LIN {X 0,Y 560.526,Z 804.621,A -85,B 0,C 180,E1 21133.416,E2 21133.416} C_VEL
LIN {X 0,Y 560.837,Z 791.782,A -85,B 0,C 180,E1 21131.497,E2 21131.497} C_VEL
LIN {X 0,Y 561.234,Z 777.649,A -85,B 0,C 180,E1 21129.671,E2 21129.671} C_VEL
LIN {X 0,Y 561.729,Z 761.82,A -85,B 0,C 180,E1 21127.907,E2 21127.907} C_VEL
LIN {X 0,Y 562.275,Z 745.057,A -85,B 0,C 180,E1 21126.303,E2 21126.303} C_VEL
LIN {X 0,Y 562.895,Z 726.381,A -85,B 0,C 180,E1 21124.766,E2 21124.766} C_VEL
LIN {X 0,Y 563.513,Z 707.517,A -85,B 0,C 180,E1 21123.439,E2 21123.439} C_VEL
LIN {X 0,Y 564.133,Z 687.731,A -85,B 0,C 180,E1 21122.273,E2 21122.273} C_VEL
LIN {X 0,Y 564.708,Z 667.025,A -85,B 0,C 180,E1 21121.267,E2 21121.267} C_VEL
LIN {X 0,Y 565.266,Z 645.641,A -85,B 0,C 180,E1 21120.436,E2 21120.436} C_VEL
LIN {X 0,Y 565.671,Z 624.866,A -85,B 0,C 180,E1 21119.819,E2 21119.819} C_VEL
LIN {X 0,Y 565.989,Z 603.229,A -85,B 0,C 180,E1 21119.371,E2 21119.371} C_VEL
LIN {X 0,Y 567.351,Z 377.021,A -85,B 0,C 180,E1 21116.119,E2 21116.119} C_VEL
LIN {X 0,Y 567.583,Z 309.479,A -85,B 0,C 180,E1 21115.121,E2 21115.121} C_VEL
LIN {X 0,Y 566.29,Z 301.611,A -85,B 0,C 180,E1 21114.889,E2 21114.889} C_VEL
LIN {X 0,Y 567.231,Z 259.014,A -85,B 0,C 180,E1 21112.198,E2 21112.198} C_VEL
LIN {X 0,Y 561.642,Z 246.538,A -85,B 0,C 180,E1 21110.913,E2 21110.913} C_VEL
LIN {X 0,Y 560.282,Z 243.194,A -85,B 0,C 180,E1 21110.524,E2 21110.524} C_VEL
LIN {X 0,Y 560.279,Z 242.946,A -85,B 0,C 180,E1 21107.479,E2 21107.479} C_VEL
LIN {X 0,Y 560.273,Z 242.948,A -85,B 0,C 180,E1 21104.106,E2 21104.106} C_VEL
LIN {X 0,Y 560.259,Z 242.944,A -85,B 0,C 180,E1 21100.782,E2 21100.782} C_VEL
LIN {X 0,Y 560.272,Z 242.944,A -85,B 0,C 180,E1 21097.485,E2 21097.485} C_VEL
LIN {X 0,Y 560.274,Z 242.947,A -85,B 0,C 180,E1 21094.1,E2 21094.1} C_VEL
LIN {X 0,Y 560.266,Z 242.942,A -85,B 0,C 180,E1 21090.691,E2 21090.691} C_VEL
LIN {X 0,Y 560.266,Z 242.943,A -85,B 0,C 180,E1 21087.415,E2 21087.415} C_VEL
LIN {X 0,Y 560.278,Z 242.946,A -85,B 0,C 180,E1 21084.01,E2 21084.01} C_VEL
LIN {X 0,Y 560.276,Z 242.939,A -85,B 0,C 180,E1 21080.693,E2 21080.693} C_VEL
LIN {X 0,Y 560.256,Z 242.942,A -85,B 0,C 180,E1 21077.34,E2 21077.34} C_VEL
LIN {X 0,Y 560.28,Z 242.945,A -85,B 0,C 180,E1 21074.047,E2 21074.047} C_VEL
LIN {X 0,Y 560.278,Z 242.937,A -85,B 0,C 180,E1 21070.697,E2 21070.697} C_VEL
LIN {X 0,Y 560.249,Z 242.945,A -85,B 0,C 180,E1 21067.383,E2 21067.383} C_VEL
LIN {X 0,Y 560.279,Z 242.944,A -85,B 0,C 180,E1 21064.094,E2 21064.094} C_VEL
LIN {X 0,Y 560.256,Z 242.941,A -85,B 0,C 180,E1 21060.819,E2 21060.819} C_VEL
LIN {X 0,Y 560.244,Z 242.947,A -85,B 0,C 180,E1 21057.444,E2 21057.444} C_VEL
LIN {X 0,Y 560.283,Z 242.944,A -85,B 0,C 180,E1 21054.163,E2 21054.163} C_VEL
LIN {X 0,Y 560.233,Z 242.945,A -85,B 0,C 180,E1 21050.965,E2 21050.965} C_VEL
LIN {X 0,Y 560.252,Z 242.949,A -85,B 0,C 180,E1 21047.635,E2 21047.635} C_VEL
LIN {X 0,Y 560.255,Z 242.945,A -85,B 0,C 180,E1 21044.474,E2 21044.474} C_VEL
LIN {X 0,Y 560.22,Z 242.949,A -85,B 0,C 180,E1 21041.154,E2 21041.154} C_VEL
LIN {X 0,Y 560.285,Z 242.943,A -85,B 0,C 180,E1 21037.992,E2 21037.992} C_VEL
LIN {X 0,Y 560.252,Z 242.943,A -85,B 0,C 180,E1 21036.326,E2 21036.326} C_VEL
LIN {X 0,Y 559.308,Z 243.067,A -85,B 0,C 180,E1 21035.538,E2 21035.538} C_VEL
LIN {X 0,Y 552.806,Z 243.877,A -85,B 0,C 180,E1 21033.327,E2 21033.327} C_VEL
LIN {X 0,Y 552.275,Z 243.943,A -85,B 0,C 180,E1 21032.75,E2 21032.75} C_VEL
LIN {X 0,Y 552.312,Z 244.188,A -85,B 0,C 180,E1 21031.274,E2 21031.274} C_VEL
LIN {X 0,Y 557.253,Z 257.483,A -85,B 0,C 180,E1 21029.724,E2 21029.724} C_VEL
LIN {X 0,Y 557.944,Z 259.928,A -85,B 0,C 180,E1 21029.468,E2 21029.468} C_VEL
LIN {X 0,Y 556.963,Z 299.293,A -85,B 0,C 180,E1 21026.434,E2 21026.434} C_VEL
LIN {X 0,Y 558.759,Z 310.135,A -85,B 0,C 180,E1 21026.153,E2 21026.153} C_VEL
LIN {X 0,Y 557.351,Z 546.952,A -85,B 0,C 180,E1 21022.833,E2 21022.833} C_VEL
LIN {X 0,Y 557.1,Z 568.52,A -85,B 0,C 180,E1 21022.453,E2 21022.453} C_VEL
LIN {X 0,Y 556.693,Z 589.412,A -85,B 0,C 180,E1 21021.889,E2 21021.889} C_VEL
LIN {X 0,Y 556.205,Z 610.238,A -85,B 0,C 180,E1 21021.113,E2 21021.113} C_VEL
LIN {X 0,Y 555.666,Z 629.254,A -85,B 0,C 180,E1 21020.206,E2 21020.206} C_VEL
LIN {X 0,Y 555.086,Z 647.945,A -85,B 0,C 180,E1 21019.107,E2 21019.107} C_VEL
LIN {X 0,Y 554.471,Z 666.341,A -85,B 0,C 180,E1 21017.796,E2 21017.796} C_VEL
LIN {X 0,Y 553.907,Z 683.018,A -85,B 0,C 180,E1 21016.374,E2 21016.374} C_VEL
LIN {X 0,Y 553.405,Z 698.157,A -85,B 0,C 180,E1 21014.857,E2 21014.857} C_VEL
LIN {X 0,Y 552.977,Z 712.083,A -85,B 0,C 180,E1 21013.226,E2 21013.226} C_VEL
LIN {X 0,Y 552.603,Z 725.775,A -85,B 0,C 180,E1 21011.335,E2 21011.335} C_VEL
LIN {X 0,Y 552.324,Z 737.233,A -85,B 0,C 180,E1 21009.451,E2 21009.451} C_VEL
LIN {X 0,Y 552.14,Z 747.227,A -85,B 0,C 180,E1 21007.479,E2 21007.479} C_VEL
LIN {X 0,Y 552.015,Z 755.724,A -85,B 0,C 180,E1 21005.408,E2 21005.408} C_VEL
LIN {X 0,Y 551.945,Z 762.22,A -85,B 0,C 180,E1 21003.376,E2 21003.376} C_VEL
LIN {X 0,Y 551.914,Z 767.119,A -85,B 0,C 180,E1 21001.329,E2 21001.329} C_VEL
LIN {X 0,Y 551.906,Z 770.434,A -85,B 0,C 180,E1 20999.285,E2 20999.285} C_VEL
LIN {X 0,Y 551.907,Z 772.23,A -85,B 0,C 180,E1 20997.165,E2 20997.165} C_VEL
LIN {X 0,Y 551.911,Z 772.317,A -85,B 0,C 180,E1 20995.071,E2 20995.071} C_VEL
LIN {X 0,Y 551.911,Z 770.762,A -85,B 0,C 180,E1 20992.924,E2 20992.924} C_VEL
LIN {X 0,Y 551.915,Z 767.546,A -85,B 0,C 180,E1 20990.799,E2 20990.799} C_VEL
LIN {X 0,Y 551.938,Z 763.025,A -85,B 0,C 180,E1 20988.812,E2 20988.812} C_VEL
LIN {X 0,Y 551.997,Z 756.558,A -85,B 0,C 180,E1 20986.739,E2 20986.739} C_VEL
LIN {X 0,Y 552.111,Z 748.635,A -85,B 0,C 180,E1 20984.754,E2 20984.754} C_VEL
LIN {X 0,Y 552.292,Z 738.872,A -85,B 0,C 180,E1 20982.761,E2 20982.761} C_VEL
LIN {X 0,Y 552.552,Z 727.572,A -85,B 0,C 180,E1 20980.848,E2 20980.848} C_VEL
LIN {X 0,Y 552.889,Z 714.988,A -85,B 0,C 180,E1 20979.053,E2 20979.053} C_VEL
LIN {X 0,Y 553.317,Z 701.127,A -85,B 0,C 180,E1 20977.372,E2 20977.372} C_VEL
LIN {X 0,Y 553.821,Z 685.347,A -85,B 0,C 180,E1 20975.752,E2 20975.752} C_VEL
LIN {X 0,Y 554.388,Z 668.562,A -85,B 0,C 180,E1 20974.293,E2 20974.293} C_VEL
LIN {X 0,Y 554.989,Z 650.803,A -85,B 0,C 180,E1 20972.996,E2 20972.996} C_VEL
LIN {X 0,Y 555.576,Z 632.057,A -85,B 0,C 180,E1 20971.857,E2 20971.857} C_VEL
LIN {X 0,Y 556.151,Z 612.112,A -85,B 0,C 180,E1 20970.877,E2 20970.877} C_VEL
LIN {X 0,Y 556.643,Z 592.022,A -85,B 0,C 180,E1 20970.104,E2 20970.104} C_VEL
LIN {X 0,Y 557.074,Z 571.838,A -85,B 0,C 180,E1 20969.529,E2 20969.529} C_VEL
LIN {X 0,Y 557.327,Z 550.613,A -85,B 0,C 180,E1 20969.129,E2 20969.129} C_VEL
LIN {X 0,Y 558.765,Z 309.101,A -85,B 0,C 180,E1 20965.742,E2 20965.742} C_VEL
LIN {X 0,Y 556.955,Z 299.19,A -85,B 0,C 180,E1 20965.471,E2 20965.471} C_VEL
LIN {X 0,Y 557.923,Z 259.153,A -85,B 0,C 180,E1 20962.38,E2 20962.38} C_VEL
LIN {X 0,Y 552.377,Z 244.203,A -85,B 0,C 180,E1 20960.678,E2 20960.678} C_VEL
LIN {X 0,Y 552.338,Z 243.928,A -85,B 0,C 180,E1 20958.833,E2 20958.833} C_VEL
LIN {X 0,Y 552.32,Z 243.926,A -85,B 0,C 180,E1 20955.427,E2 20955.427} C_VEL
LIN {X 0,Y 552.335,Z 243.92,A -85,B 0,C 180,E1 20952.078,E2 20952.078} C_VEL
LIN {X 0,Y 552.342,Z 243.929,A -85,B 0,C 180,E1 20948.664,E2 20948.664} C_VEL
LIN {X 0,Y 552.318,Z 243.93,A -85,B 0,C 180,E1 20945.282,E2 20945.282} C_VEL
LIN {X 0,Y 552.337,Z 243.934,A -85,B 0,C 180,E1 20941.924,E2 20941.924} C_VEL
LIN {X 0,Y 552.34,Z 243.927,A -85,B 0,C 180,E1 20938.494,E2 20938.494} C_VEL
LIN {X 0,Y 552.317,Z 243.93,A -85,B 0,C 180,E1 20935.088,E2 20935.088} C_VEL
LIN {X 0,Y 552.338,Z 243.935,A -85,B 0,C 180,E1 20931.752,E2 20931.752} C_VEL
LIN {X 0,Y 552.339,Z 243.928,A -85,B 0,C 180,E1 20928.369,E2 20928.369} C_VEL
LIN {X 0,Y 552.317,Z 243.932,A -85,B 0,C 180,E1 20924.944,E2 20924.944} C_VEL
LIN {X 0,Y 552.338,Z 243.933,A -85,B 0,C 180,E1 20921.617,E2 20921.617} C_VEL
LIN {X 0,Y 552.338,Z 243.928,A -85,B 0,C 180,E1 20918.223,E2 20918.223} C_VEL
LIN {X 0,Y 552.319,Z 243.933,A -85,B 0,C 180,E1 20914.892,E2 20914.892} C_VEL
LIN {X 0,Y 552.338,Z 243.932,A -85,B 0,C 180,E1 20911.543,E2 20911.543} C_VEL
LIN {X 0,Y 552.328,Z 243.929,A -85,B 0,C 180,E1 20908.194,E2 20908.194} C_VEL
LIN {X 0,Y 552.32,Z 243.932,A -85,B 0,C 180,E1 20904.832,E2 20904.832} C_VEL
LIN {X 0,Y 552.338,Z 243.932,A -85,B 0,C 180,E1 20901.498,E2 20901.498} C_VEL
LIN {X 0,Y 552.321,Z 243.928,A -85,B 0,C 180,E1 20898.127,E2 20898.127} C_VEL
LIN {X 0,Y 552.319,Z 243.927,A -85,B 0,C 180,E1 20894.68,E2 20894.68} C_VEL
LIN {X 0,Y 552.338,Z 243.931,A -85,B 0,C 180,E1 20891.379,E2 20891.379} C_VEL
LIN {X 0,Y 552.316,Z 243.925,A -85,B 0,C 180,E1 20888.026,E2 20888.026} C_VEL
LIN {X 0,Y 552.322,Z 243.932,A -85,B 0,C 180,E1 20884.568,E2 20884.568} C_VEL
LIN {X 0,Y 552.337,Z 243.929,A -85,B 0,C 180,E1 20881.244,E2 20881.244} C_VEL
LIN {X 0,Y 552.31,Z 243.926,A -85,B 0,C 180,E1 20878.028,E2 20878.028} C_VEL
LIN {X 0,Y 552.333,Z 243.935,A -85,B 0,C 180,E1 20874.626,E2 20874.626} C_VEL
LIN {X 0,Y 552.341,Z 243.926,A -85,B 0,C 180,E1 20871.245,E2 20871.245} C_VEL
LIN {X 0,Y 552.308,Z 243.926,A -85,B 0,C 180,E1 20867.983,E2 20867.983} C_VEL
LIN {X 0,Y 552.341,Z 243.937,A -85,B 0,C 180,E1 20864.674,E2 20864.674} C_VEL
LIN {X 0,Y 552.332,Z 243.929,A -85,B 0,C 180,E1 20861.311,E2 20861.311} C_VEL
LIN {X 0,Y 552.309,Z 243.934,A -85,B 0,C 180,E1 20857.95,E2 20857.95} C_VEL
LIN {X 0,Y 552.338,Z 243.93,A -85,B 0,C 180,E1 20854.709,E2 20854.709} C_VEL
LIN {X 0,Y 552.314,Z 243.927,A -85,B 0,C 180,E1 20851.398,E2 20851.398} C_VEL
LIN {X 0,Y 552.316,Z 243.934,A -85,B 0,C 180,E1 20847.966,E2 20847.966} C_VEL
LIN {X 0,Y 552.341,Z 243.931,A -85,B 0,C 180,E1 20844.6,E2 20844.6} C_VEL
LIN {X 0,Y 552.312,Z 243.933,A -85,B 0,C 180,E1 20841.281,E2 20841.281} C_VEL
LIN {X 0,Y 552.313,Z 243.934,A -85,B 0,C 180,E1 20837.807,E2 20837.807} C_VEL
LIN {X 0,Y 552.342,Z 243.928,A -85,B 0,C 180,E1 20834.469,E2 20834.469} C_VEL
LIN {X 0,Y 552.309,Z 243.917,A -85,B 0,C 180,E1 20831.141,E2 20831.141} C_VEL
LIN {X 0,Y 552.377,Z 244.171,A -85,B 0,C 180,E1 20830.084,E2 20830.084} C_VEL
LIN {X 0,Y 553.624,Z 247.426,A -85,B 0,C 180,E1 20829.703,E2 20829.703} C_VEL
LIN {X 0,Y 560.495,Z 262.477,A -85,B 0,C 180,E1 20828.106,E2 20828.106} C_VEL
LIN {X 0,Y 559.572,Z 302.658,A -85,B 0,C 180,E1 20825.56,E2 20825.56} C_VEL
LIN {X 0,Y 561.188,Z 313.338,A -85,B 0,C 180,E1 20825.276,E2 20825.276} C_VEL
LIN {X 0,Y 559.615,Z 532.328,A -85,B 0,C 180,E1 20822.08,E2 20822.08} C_VEL
LIN {X 0,Y 559.046,Z 609.244,A -85,B 0,C 180,E1 20820.946,E2 20820.946} C_VEL
LIN {X 0,Y 558.582,Z 630.7,A -85,B 0,C 180,E1 20820.438,E2 20820.438} C_VEL
LIN {X 0,Y 558.05,Z 652.597,A -85,B 0,C 180,E1 20819.721,E2 20819.721} C_VEL
LIN {X 0,Y 557.44,Z 673.421,A -85,B 0,C 180,E1 20818.847,E2 20818.847} C_VEL
LIN {X 0,Y 556.703,Z 693.771,A -85,B 0,C 180,E1 20817.778,E2 20817.778} C_VEL
LIN {X 0,Y 555.95,Z 714.163,A -85,B 0,C 180,E1 20816.487,E2 20816.487} C_VEL
LIN {X 0,Y 555.199,Z 733.164,A -85,B 0,C 180,E1 20815.062,E2 20815.062} C_VEL
LIN {X 0,Y 554.505,Z 751.125,A -85,B 0,C 180,E1 20813.483,E2 20813.483} C_VEL
LIN {X 0,Y 553.868,Z 767.711,A -85,B 0,C 180,E1 20811.774,E2 20811.774} C_VEL
LIN {X 0,Y 553.321,Z 782.881,A -85,B 0,C 180,E1 20809.968,E2 20809.968} C_VEL
LIN {X 0,Y 552.873,Z 797.052,A -85,B 0,C 180,E1 20808.013,E2 20808.013} C_VEL
LIN {X 0,Y 552.514,Z 809.742,A -85,B 0,C 180,E1 20805.965,E2 20805.965} C_VEL
LIN {X 0,Y 552.258,Z 820.339,A -85,B 0,C 180,E1 20803.932,E2 20803.932} C_VEL
LIN {X 0,Y 552.085,Z 830.073,A -85,B 0,C 180,E1 20801.702,E2 20801.702} C_VEL
LIN {X 0,Y 551.99,Z 837.94,A -85,B 0,C 180,E1 20799.486,E2 20799.486} C_VEL
LIN {X 0,Y 551.939,Z 843.91,A -85,B 0,C 180,E1 20797.284,E2 20797.284} C_VEL
LIN {X 0,Y 551.92,Z 848.466,A -85,B 0,C 180,E1 20794.987,E2 20794.987} C_VEL
LIN {X 0,Y 551.909,Z 851.235,A -85,B 0,C 180,E1 20792.803,E2 20792.803} C_VEL
LIN {X 0,Y 551.898,Z 852.373,A -85,B 0,C 180,E1 20790.622,E2 20790.622} C_VEL
LIN {X 0,Y 551.899,Z 852.014,A -85,B 0,C 180,E1 20788.338,E2 20788.338} C_VEL
LIN {X 0,Y 551.905,Z 850.22,A -85,B 0,C 180,E1 20786.26,E2 20786.26} C_VEL
LIN {X 0,Y 551.922,Z 846.601,A -85,B 0,C 180,E1 20783.968,E2 20783.968} C_VEL
LIN {X 0,Y 551.965,Z 841.58,A -85,B 0,C 180,E1 20781.771,E2 20781.771} C_VEL
LIN {X 0,Y 552.026,Z 835.108,A -85,B 0,C 180,E1 20779.669,E2 20779.669} C_VEL
LIN {X 0,Y 552.147,Z 826.54,A -85,B 0,C 180,E1 20777.435,E2 20777.435} C_VEL
LIN {X 0,Y 552.352,Z 816.683,A -85,B 0,C 180,E1 20775.319,E2 20775.319} C_VEL
LIN {X 0,Y 552.633,Z 805.264,A -85,B 0,C 180,E1 20773.28,E2 20773.28} C_VEL
LIN {X 0,Y 553.028,Z 791.783,A -85,B 0,C 180,E1 20771.226,E2 20771.226} C_VEL
LIN {X 0,Y 553.515,Z 777.378,A -85,B 0,C 180,E1 20769.342,E2 20769.342} C_VEL
LIN {X 0,Y 554.098,Z 761.611,A -85,B 0,C 180,E1 20767.563,E2 20767.563} C_VEL
LIN {X 0,Y 554.756,Z 744.446,A -85,B 0,C 180,E1 20765.905,E2 20765.905} C_VEL
LIN {X 0,Y 555.498,Z 725.729,A -85,B 0,C 180,E1 20764.354,E2 20764.354} C_VEL
LIN {X 0,Y 556.232,Z 706.63,A -85,B 0,C 180,E1 20763.006,E2 20763.006} C_VEL
LIN {X 0,Y 556.963,Z 686.724,A -85,B 0,C 180,E1 20761.826,E2 20761.826} C_VEL
LIN {X 0,Y 557.638,Z 666.253,A -85,B 0,C 180,E1 20760.833,E2 20760.833} C_VEL
LIN {X 0,Y 558.264,Z 644.537,A -85,B 0,C 180,E1 20759.99,E2 20759.99} C_VEL
LIN {X 0,Y 558.787,Z 623.271,A -85,B 0,C 180,E1 20759.362,E2 20759.362} C_VEL
LIN {X 0,Y 559.111,Z 601.699,A -85,B 0,C 180,E1 20758.926,E2 20758.926} C_VEL
LIN {X 0,Y 560.691,Z 379.462,A -85,B 0,C 180,E1 20755.698,E2 20755.698} C_VEL
LIN {X 0,Y 561.012,Z 310.948,A -85,B 0,C 180,E1 20754.674,E2 20754.674} C_VEL
LIN {X 0,Y 559.48,Z 301.734,A -85,B 0,C 180,E1 20754.404,E2 20754.404} C_VEL
LIN {X 0,Y 560.438,Z 262.344,A -85,B 0,C 180,E1 20751.881,E2 20751.881} C_VEL
LIN {X 0,Y 553.279,Z 246.849,A -85,B 0,C 180,E1 20750.227,E2 20750.227} C_VEL
LIN {X 0,Y 552.374,Z 244.151,A -85,B 0,C 180,E1 20749.912,E2 20749.912} C_VEL
LIN {X 0,Y 552.312,Z 243.935,A -85,B 0,C 180,E1 20746.676,E2 20746.676} C_VEL
LIN {X 0,Y 552.339,Z 243.924,A -85,B 0,C 180,E1 20743.321,E2 20743.321} C_VEL
LIN {X 0,Y 552.34,Z 243.936,A -85,B 0,C 180,E1 20739.866,E2 20739.866} C_VEL
LIN {X 0,Y 552.321,Z 243.934,A -85,B 0,C 180,E1 20736.508,E2 20736.508} C_VEL
LIN {X 0,Y 552.34,Z 243.93,A -85,B 0,C 180,E1 20733.14,E2 20733.14} C_VEL
LIN {X 0,Y 552.333,Z 243.932,A -85,B 0,C 180,E1 20729.666,E2 20729.666} C_VEL
LIN {X 0,Y 552.33,Z 243.933,A -85,B 0,C 180,E1 20726.329,E2 20726.329} C_VEL
LIN {X 0,Y 552.343,Z 243.927,A -85,B 0,C 180,E1 20722.905,E2 20722.905} C_VEL
LIN {X 0,Y 552.324,Z 243.935,A -85,B 0,C 180,E1 20719.567,E2 20719.567} C_VEL
LIN {X 0,Y 552.337,Z 243.933,A -85,B 0,C 180,E1 20716.188,E2 20716.188} C_VEL
LIN {X 0,Y 552.339,Z 243.929,A -85,B 0,C 180,E1 20712.759,E2 20712.759} C_VEL
LIN {X 0,Y 552.312,Z 243.934,A -85,B 0,C 180,E1 20709.378,E2 20709.378} C_VEL
LIN {X 0,Y 552.341,Z 243.936,A -85,B 0,C 180,E1 20706.028,E2 20706.028} C_VEL
LIN {X 0,Y 552.336,Z 243.93,A -85,B 0,C 180,E1 20702.595,E2 20702.595} C_VEL
LIN {X 0,Y 552.3,Z 243.933,A -85,B 0,C 180,E1 20699.275,E2 20699.275} C_VEL
LIN {X 0,Y 552.338,Z 243.935,A -85,B 0,C 180,E1 20695.953,E2 20695.953} C_VEL
LIN {X 0,Y 552.309,Z 243.93,A -85,B 0,C 180,E1 20692.721,E2 20692.721} C_VEL
LIN {X 0,Y 552.296,Z 243.937,A -85,B 0,C 180,E1 20689.36,E2 20689.36} C_VEL
LIN {X 0,Y 552.348,Z 243.935,A -85,B 0,C 180,E1 20686.07,E2 20686.07} C_VEL
LIN {X 0,Y 552.287,Z 243.936,A -85,B 0,C 180,E1 20682.838,E2 20682.838} C_VEL
LIN {X 0,Y 552.293,Z 243.94,A -85,B 0,C 180,E1 20679.44,E2 20679.44} C_VEL
LIN {X 0,Y 552.315,Z 243.931,A -85,B 0,C 180,E1 20676.305,E2 20676.305} C_VEL
LIN {X 0,Y 552.274,Z 243.943,A -85,B 0,C 180,E1 20673.09,E2 20673.09} C_VEL
LIN {X 0,Y 552.275,Z 243.943,A -85,B 0,C 180,E1 20672.75,E2 20672.75} C_VEL
LIN {X 0,Y 552.203,Z 244.856,A -85,B 0,C 180,E1 20672.128,E2 20672.128} C_VEL
LIN {X 0,Y 551.96,Z 247.757,A -85,B 0,C 180,E1 20671.441,E2 20671.441} C_VEL
LIN {X 0,Y 551.548,Z 253.184,A -85,B 0,C 180,E1 20670.684,E2 20670.684} C_VEL
LIN {X 0,Y 551.05,Z 261.64,A -85,B 0,C 180,E1 20669.859,E2 20669.859} C_VEL
LIN {X 0,Y 550.975,Z 263.457,A -85,B 0,C 180,E1 20669.708,E2 20669.708} C_VEL
LIN {X 0,Y 549.764,Z 298.397,A -85,B 0,C 180,E1 20666.935,E2 20666.935} C_VEL
LIN {X 0,Y 550.294,Z 302.24,A -85,B 0,C 180,E1 20666.785,E2 20666.785} C_VEL
LIN {X 0,Y 551.836,Z 311.511,A -85,B 0,C 180,E1 20666.552,E2 20666.552} C_VEL
LIN {X 0,Y 550.207,Z 548.465,A -85,B 0,C 180,E1 20663.189,E2 20663.189} C_VEL
LIN {X 0,Y 549.916,Z 569.449,A -85,B 0,C 180,E1 20662.806,E2 20662.806} C_VEL
LIN {X 0,Y 549.453,Z 589.959,A -85,B 0,C 180,E1 20662.239,E2 20662.239} C_VEL
LIN {X 0,Y 548.903,Z 610.312,A -85,B 0,C 180,E1 20661.468,E2 20661.468} C_VEL
LIN {X 0,Y 548.268,Z 629.602,A -85,B 0,C 180,E1 20660.534,E2 20660.534} C_VEL
LIN {X 0,Y 547.601,Z 648.163,A -85,B 0,C 180,E1 20659.427,E2 20659.427} C_VEL
LIN {X 0,Y 546.924,Z 665.931,A -85,B 0,C 180,E1 20658.145,E2 20658.145} C_VEL
LIN {X 0,Y 546.262,Z 682.71,A -85,B 0,C 180,E1 20656.701,E2 20656.701} C_VEL
LIN {X 0,Y 545.665,Z 698.158,A -85,B 0,C 180,E1 20655.135,E2 20655.135} C_VEL
LIN {X 0,Y 545.149,Z 712.524,A -85,B 0,C 180,E1 20653.425,E2 20653.425} C_VEL
LIN {X 0,Y 544.713,Z 726.171,A -85,B 0,C 180,E1 20651.502,E2 20651.502} C_VEL
LIN {X 0,Y 544.381,Z 737.927,A -85,B 0,C 180,E1 20649.522,E2 20649.522} C_VEL
LIN {X 0,Y 544.173,Z 747.479,A -85,B 0,C 180,E1 20647.591,E2 20647.591} C_VEL
LIN {X 0,Y 544.034,Z 755.913,A -85,B 0,C 180,E1 20645.497,E2 20645.497} C_VEL
LIN {X 0,Y 543.948,Z 762.632,A -85,B 0,C 180,E1 20643.341,E2 20643.341} C_VEL
LIN {X 0,Y 543.914,Z 767.474,A -85,B 0,C 180,E1 20641.225,E2 20641.225} C_VEL
LIN {X 0,Y 543.908,Z 770.758,A -85,B 0,C 180,E1 20639.034,E2 20639.034} C_VEL
LIN {X 0,Y 543.913,Z 772.309,A -85,B 0,C 180,E1 20636.887,E2 20636.887} C_VEL
LIN {X 0,Y 543.913,Z 772.245,A -85,B 0,C 180,E1 20634.759,E2 20634.759} C_VEL
LIN {X 0,Y 543.912,Z 770.455,A -85,B 0,C 180,E1 20632.595,E2 20632.595} C_VEL
LIN {X 0,Y 543.92,Z 767.223,A -85,B 0,C 180,E1 20630.556,E2 20630.556} C_VEL
LIN {X 0,Y 543.952,Z 762.24,A -85,B 0,C 180,E1 20628.432,E2 20628.432} C_VEL
LIN {X 0,Y 544.04,Z 755.61,A -85,B 0,C 180,E1 20626.332,E2 20626.332} C_VEL
LIN {X 0,Y 544.182,Z 747.199,A -85,B 0,C 180,E1 20624.254,E2 20624.254} C_VEL
LIN {X 0,Y 544.392,Z 737.423,A -85,B 0,C 180,E1 20622.294,E2 20622.294} C_VEL
LIN {X 0,Y 544.717,Z 725.888,A -85,B 0,C 180,E1 20620.364,E2 20620.364} C_VEL
LIN {X 0,Y 545.13,Z 712.985,A -85,B 0,C 180,E1 20618.545,E2 20618.545} C_VEL
LIN {X 0,Y 545.646,Z 698.78,A -85,B 0,C 180,E1 20616.842,E2 20616.842} C_VEL
LIN {X 0,Y 546.245,Z 683.193,A -85,B 0,C 180,E1 20615.252,E2 20615.252} C_VEL
LIN {X 0,Y 546.919,Z 666.062,A -85,B 0,C 180,E1 20613.775,E2 20613.775} C_VEL
LIN {X 0,Y 547.616,Z 647.823,A -85,B 0,C 180,E1 20612.46,E2 20612.46} C_VEL
LIN {X 0,Y 548.282,Z 629.306,A -85,B 0,C 180,E1 20611.36,E2 20611.36} C_VEL
LIN {X 0,Y 548.888,Z 610.865,A -85,B 0,C 180,E1 20610.466,E2 20610.466} C_VEL
LIN {X 0,Y 549.435,Z 590.31,A -85,B 0,C 180,E1 20609.682,E2 20609.682} C_VEL
LIN {X 0,Y 549.917,Z 569.978,A -85,B 0,C 180,E1 20609.116,E2 20609.116} C_VEL
LIN {X 0,Y 550.203,Z 548.996,A -85,B 0,C 180,E1 20608.729,E2 20608.729} C_VEL
LIN {X 0,Y 551.842,Z 310.385,A -85,B 0,C 180,E1 20605.342,E2 20605.342} C_VEL
LIN {X 0,Y 549.781,Z 299.048,A -85,B 0,C 180,E1 20605.019,E2 20605.019} C_VEL
LIN {X 0,Y 550.896,Z 262.387,A -85,B 0,C 180,E1 20602.125,E2 20602.125} C_VEL
LIN {X 0,Y 544.445,Z 245.239,A -85,B 0,C 180,E1 20600.141,E2 20600.141} C_VEL
LIN {X 0,Y 544.38,Z 244.904,A -85,B 0,C 180,E1 20599.418,E2 20599.418} C_VEL
LIN {X 0,Y 544.398,Z 244.904,A -85,B 0,C 180,E1 20596.079,E2 20596.079} C_VEL
LIN {X 0,Y 544.399,Z 244.914,A -85,B 0,C 180,E1 20592.692,E2 20592.692} C_VEL
LIN {X 0,Y 544.383,Z 244.924,A -85,B 0,C 180,E1 20589.352,E2 20589.352} C_VEL
LIN {X 0,Y 544.394,Z 244.903,A -85,B 0,C 180,E1 20586.054,E2 20586.054} C_VEL
LIN {X 0,Y 544.397,Z 244.919,A -85,B 0,C 180,E1 20582.669,E2 20582.669} C_VEL
LIN {X 0,Y 544.382,Z 244.922,A -85,B 0,C 180,E1 20579.265,E2 20579.265} C_VEL
LIN {X 0,Y 544.398,Z 244.923,A -85,B 0,C 180,E1 20575.924,E2 20575.924} C_VEL
LIN {X 0,Y 544.394,Z 244.918,A -85,B 0,C 180,E1 20572.505,E2 20572.505} C_VEL
LIN {X 0,Y 544.384,Z 244.924,A -85,B 0,C 180,E1 20569.169,E2 20569.169} C_VEL
LIN {X 0,Y 544.397,Z 244.918,A -85,B 0,C 180,E1 20565.889,E2 20565.889} C_VEL
LIN {X 0,Y 544.386,Z 244.918,A -85,B 0,C 180,E1 20562.522,E2 20562.522} C_VEL
LIN {X 0,Y 544.383,Z 244.924,A -85,B 0,C 180,E1 20559.023,E2 20559.023} C_VEL
LIN {X 0,Y 544.397,Z 244.915,A -85,B 0,C 180,E1 20555.731,E2 20555.731} C_VEL
LIN {X 0,Y 544.383,Z 244.917,A -85,B 0,C 180,E1 20552.345,E2 20552.345} C_VEL
LIN {X 0,Y 544.384,Z 244.924,A -85,B 0,C 180,E1 20548.883,E2 20548.883} C_VEL
LIN {X 0,Y 544.398,Z 244.918,A -85,B 0,C 180,E1 20545.568,E2 20545.568} C_VEL
LIN {X 0,Y 544.38,Z 244.92,A -85,B 0,C 180,E1 20542.231,E2 20542.231} C_VEL
LIN {X 0,Y 544.382,Z 244.922,A -85,B 0,C 180,E1 20538.748,E2 20538.748} C_VEL
LIN {X 0,Y 544.4,Z 244.92,A -85,B 0,C 180,E1 20535.378,E2 20535.378} C_VEL
LIN {X 0,Y 544.377,Z 244.919,A -85,B 0,C 180,E1 20532.085,E2 20532.085} C_VEL
LIN {X 0,Y 544.384,Z 244.917,A -85,B 0,C 180,E1 20528.661,E2 20528.661} C_VEL
LIN {X 0,Y 544.4,Z 244.92,A -85,B 0,C 180,E1 20525.374,E2 20525.374} C_VEL
LIN {X 0,Y 544.375,Z 244.917,A -85,B 0,C 180,E1 20521.999,E2 20521.999} C_VEL
LIN {X 0,Y 544.391,Z 244.919,A -85,B 0,C 180,E1 20518.631,E2 20518.631} C_VEL
LIN {X 0,Y 544.402,Z 244.918,A -85,B 0,C 180,E1 20515.258,E2 20515.258} C_VEL
LIN {X 0,Y 544.371,Z 244.917,A -85,B 0,C 180,E1 20511.975,E2 20511.975} C_VEL
LIN {X 0,Y 544.396,Z 244.919,A -85,B 0,C 180,E1 20508.558,E2 20508.558} C_VEL
LIN {X 0,Y 544.405,Z 244.919,A -85,B 0,C 180,E1 20505.1,E2 20505.1} C_VEL
LIN {X 0,Y 544.371,Z 244.921,A -85,B 0,C 180,E1 20501.724,E2 20501.724} C_VEL
LIN {X 0,Y 544.391,Z 244.922,A -85,B 0,C 180,E1 20498.329,E2 20498.329} C_VEL
LIN {X 0,Y 544.403,Z 244.916,A -85,B 0,C 180,E1 20495.012,E2 20495.012} C_VEL
LIN {X 0,Y 544.367,Z 244.918,A -85,B 0,C 180,E1 20491.713,E2 20491.713} C_VEL
LIN {X 0,Y 544.403,Z 244.922,A -85,B 0,C 180,E1 20488.437,E2 20488.437} C_VEL
LIN {X 0,Y 544.397,Z 244.917,A -85,B 0,C 180,E1 20484.996,E2 20484.996} C_VEL
LIN {X 0,Y 544.368,Z 244.924,A -85,B 0,C 180,E1 20481.624,E2 20481.624} C_VEL
LIN {X 0,Y 544.402,Z 244.924,A -85,B 0,C 180,E1 20478.328,E2 20478.328} C_VEL
LIN {X 0,Y 544.382,Z 244.911,A -85,B 0,C 180,E1 20474.998,E2 20474.998} C_VEL
LIN {X 0,Y 544.367,Z 244.9,A -85,B 0,C 180,E1 20471.621,E2 20471.621} C_VEL
LIN {X 0,Y 544.44,Z 245.141,A -85,B 0,C 180,E1 20470.67,E2 20470.67} C_VEL
LIN {X 0,Y 545.779,Z 248.516,A -85,B 0,C 180,E1 20470.269,E2 20470.269} C_VEL
LIN {X 0,Y 553.802,Z 266.258,A -85,B 0,C 180,E1 20468.393,E2 20468.393} C_VEL
LIN {X 0,Y 552.804,Z 302.684,A -85,B 0,C 180,E1 20466.062,E2 20466.062} C_VEL
LIN {X 0,Y 554.644,Z 314.755,A -85,B 0,C 180,E1 20465.734,E2 20465.734} C_VEL
LIN {X 0,Y 552.827,Z 533.496,A -85,B 0,C 180,E1 20462.504,E2 20462.504} C_VEL
LIN {X 0,Y 552.18,Z 609.244,A -85,B 0,C 180,E1 20461.374,E2 20461.374} C_VEL
LIN {X 0,Y 551.645,Z 630.83,A -85,B 0,C 180,E1 20460.858,E2 20460.858} C_VEL
LIN {X 0,Y 551.05,Z 652.52,A -85,B 0,C 180,E1 20460.141,E2 20460.141} C_VEL
LIN {X 0,Y 550.358,Z 672.381,A -85,B 0,C 180,E1 20459.304,E2 20459.304} C_VEL
LIN {X 0,Y 549.582,Z 691.72,A -85,B 0,C 180,E1 20458.292,E2 20458.292} C_VEL
LIN {X 0,Y 548.726,Z 711.65,A -85,B 0,C 180,E1 20457.045,E2 20457.045} C_VEL
LIN {X 0,Y 547.885,Z 730.773,A -85,B 0,C 180,E1 20455.626,E2 20455.626} C_VEL
LIN {X 0,Y 547.054,Z 748.712,A -85,B 0,C 180,E1 20454.051,E2 20454.051} C_VEL
LIN {X 0,Y 546.287,Z 765.685,A -85,B 0,C 180,E1 20452.319,E2 20452.319} C_VEL
LIN {X 0,Y 545.637,Z 781.182,A -85,B 0,C 180,E1 20450.486,E2 20450.486} C_VEL
LIN {X 0,Y 545.099,Z 795.638,A -85,B 0,C 180,E1 20448.5,E2 20448.5} C_VEL
LIN {X 0,Y 544.665,Z 808.471,A -85,B 0,C 180,E1 20446.42,E2 20446.42} C_VEL
LIN {X 0,Y 544.341,Z 819.821,A -85,B 0,C 180,E1 20444.248,E2 20444.248} C_VEL
LIN {X 0,Y 544.138,Z 829.259,A -85,B 0,C 180,E1 20442.09,E2 20442.09} C_VEL
LIN {X 0,Y 544.013,Z 836.888,A -85,B 0,C 180,E1 20439.947,E2 20439.947} C_VEL
LIN {X 0,Y 543.949,Z 843.148,A -85,B 0,C 180,E1 20437.71,E2 20437.71} C_VEL
LIN {X 0,Y 543.927,Z 847.826,A -85,B 0,C 180,E1 20435.484,E2 20435.484} C_VEL
LIN {X 0,Y 543.916,Z 850.787,A -85,B 0,C 180,E1 20433.266,E2 20433.266} C_VEL
LIN {X 0,Y 543.912,Z 852.306,A -85,B 0,C 180,E1 20430.947,E2 20430.947} C_VEL
LIN {X 0,Y 543.907,Z 852.237,A -85,B 0,C 180,E1 20428.735,E2 20428.735} C_VEL
LIN {X 0,Y 543.909,Z 850.559,A -85,B 0,C 180,E1 20426.521,E2 20426.521} C_VEL
LIN {X 0,Y 543.922,Z 847.218,A -85,B 0,C 180,E1 20424.196,E2 20424.196} C_VEL
LIN {X 0,Y 543.958,Z 842.633,A -85,B 0,C 180,E1 20422.075,E2 20422.075} C_VEL
LIN {X 0,Y 544.03,Z 836.173,A -85,B 0,C 180,E1 20419.837,E2 20419.837} C_VEL
LIN {X 0,Y 544.161,Z 828.426,A -85,B 0,C 180,E1 20417.692,E2 20417.692} C_VEL
LIN {X 0,Y 544.376,Z 818.771,A -85,B 0,C 180,E1 20415.534,E2 20415.534} C_VEL
LIN {X 0,Y 544.704,Z 807.188,A -85,B 0,C 180,E1 20413.359,E2 20413.359} C_VEL
LIN {X 0,Y 545.125,Z 794.866,A -85,B 0,C 180,E1 20411.388,E2 20411.388} C_VEL
LIN {X 0,Y 545.675,Z 780.314,A -85,B 0,C 180,E1 20409.401,E2 20409.401} C_VEL
LIN {X 0,Y 546.307,Z 765.158,A -85,B 0,C 180,E1 20407.623,E2 20407.623} C_VEL
LIN {X 0,Y 547.108,Z 747.479,A -85,B 0,C 180,E1 20405.834,E2 20405.834} C_VEL
LIN {X 0,Y 547.917,Z 730.02,A -85,B 0,C 180,E1 20404.316,E2 20404.316} C_VEL
LIN {X 0,Y 548.726,Z 711.653,A -85,B 0,C 180,E1 20402.955,E2 20402.955} C_VEL
LIN {X 0,Y 549.582,Z 691.721,A -85,B 0,C 180,E1 20401.708,E2 20401.708} C_VEL
LIN {X 0,Y 550.376,Z 671.623,A -85,B 0,C 180,E1 20400.662,E2 20400.662} C_VEL
LIN {X 0,Y 551.083,Z 651.726,A -85,B 0,C 180,E1 20399.829,E2 20399.829} C_VEL
LIN {X 0,Y 551.674,Z 629.585,A -85,B 0,C 180,E1 20399.107,E2 20399.107} C_VEL
LIN {X 0,Y 552.197,Z 607.826,A -85,B 0,C 180,E1 20398.602,E2 20398.602} C_VEL
LIN {X 0,Y 554.037,Z 384.564,A -85,B 0,C 180,E1 20395.306,E2 20395.306} C_VEL
LIN {X 0,Y 554.475,Z 312.436,A -85,B 0,C 180,E1 20394.217,E2 20394.217} C_VEL
LIN {X 0,Y 552.712,Z 301.611,A -85,B 0,C 180,E1 20393.893,E2 20393.893} C_VEL
LIN {X 0,Y 553.758,Z 266.113,A -85,B 0,C 180,E1 20391.594,E2 20391.594} C_VEL
LIN {X 0,Y 547.326,Z 252.072,A -85,B 0,C 180,E1 20390.109,E2 20390.109} C_VEL
LIN {X 0,Y 544.458,Z 245.269,A -85,B 0,C 180,E1 20389.373,E2 20389.373} C_VEL
LIN {X 0,Y 544.374,Z 244.913,A -85,B 0,C 180,E1 20388.856,E2 20388.856} C_VEL
LIN {X 0,Y 544.399,Z 244.916,A -85,B 0,C 180,E1 20385.592,E2 20385.592} C_VEL
LIN {X 0,Y 544.384,Z 244.916,A -85,B 0,C 180,E1 20382.239,E2 20382.239} C_VEL
LIN {X 0,Y 544.384,Z 244.922,A -85,B 0,C 180,E1 20378.779,E2 20378.779} C_VEL
LIN {X 0,Y 544.395,Z 244.922,A -85,B 0,C 180,E1 20375.478,E2 20375.478} C_VEL
LIN {X 0,Y 544.399,Z 244.924,A -85,B 0,C 180,E1 20372.059,E2 20372.059} C_VEL
LIN {X 0,Y 544.389,Z 244.918,A -85,B 0,C 180,E1 20368.606,E2 20368.606} C_VEL
LIN {X 0,Y 544.391,Z 244.92,A -85,B 0,C 180,E1 20365.221,E2 20365.221} C_VEL
LIN {X 0,Y 544.395,Z 244.924,A -85,B 0,C 180,E1 20361.778,E2 20361.778} C_VEL
LIN {X 0,Y 544.395,Z 244.922,A -85,B 0,C 180,E1 20358.416,E2 20358.416} C_VEL
LIN {X 0,Y 544.383,Z 244.919,A -85,B 0,C 180,E1 20355.119,E2 20355.119} C_VEL
LIN {X 0,Y 544.385,Z 244.921,A -85,B 0,C 180,E1 20351.657,E2 20351.657} C_VEL
LIN {X 0,Y 544.4,Z 244.923,A -85,B 0,C 180,E1 20348.237,E2 20348.237} C_VEL
LIN {X 0,Y 544.377,Z 244.918,A -85,B 0,C 180,E1 20344.953,E2 20344.953} C_VEL
LIN {X 0,Y 544.371,Z 244.923,A -85,B 0,C 180,E1 20341.474,E2 20341.474} C_VEL
LIN {X 0,Y 544.404,Z 244.92,A -85,B 0,C 180,E1 20338.212,E2 20338.212} C_VEL
LIN {X 0,Y 544.363,Z 244.922,A -85,B 0,C 180,E1 20334.943,E2 20334.943} C_VEL
LIN {X 0,Y 544.363,Z 244.925,A -85,B 0,C 180,E1 20331.445,E2 20331.445} C_VEL
LIN {X 0,Y 544.406,Z 244.923,A -85,B 0,C 180,E1 20328.131,E2 20328.131} C_VEL
LIN {X 0,Y 544.35,Z 244.925,A -85,B 0,C 180,E1 20324.882,E2 20324.882} C_VEL
LIN {X 0,Y 544.359,Z 244.928,A -85,B 0,C 180,E1 20321.474,E2 20321.474} C_VEL
LIN {X 0,Y 544.391,Z 244.925,A -85,B 0,C 180,E1 20318.224,E2 20318.224} C_VEL
LIN {X 0,Y 544.335,Z 244.927,A -85,B 0,C 180,E1 20315.011,E2 20315.011} C_VEL
LIN {X 0,Y 544.43,Z 245.169,A -85,B 0,C 180,E1 20311.838,E2 20311.838} C_VEL
LIN {X 0,Y 550.217,Z 260.475,A -85,B 0,C 180,E1 20310.019,E2 20310.019} C_VEL
LIN {X 0,Y 550.975,Z 263.457,A -85,B 0,C 180,E1 20309.708,E2 20309.708} C_VEL
LIN {X 0,Y 549.879,Z 269.811,A -85,B 0,C 180,E1 20309.258,E2 20309.258} C_VEL
LIN {X 0,Y 543.769,Z 287.639,A -85,B 0,C 180,E1 20308.224,E2 20308.224} C_VEL
LIN {X 0,Y 542.886,Z 293.11,A -85,B 0,C 180,E1 20307.831,E2 20307.831} C_VEL
LIN {X 0,Y 542.794,Z 299.97,A -85,B 0,C 180,E1 20307.321,E2 20307.321} C_VEL
LIN {X 0,Y 544.939,Z 312.828,A -85,B 0,C 180,E1 20306.962,E2 20306.962} C_VEL
LIN {X 0,Y 543.088,Z 549.357,A -85,B 0,C 180,E1 20303.563,E2 20303.563} C_VEL
LIN {X 0,Y 542.754,Z 570.473,A -85,B 0,C 180,E1 20303.166,E2 20303.166} C_VEL
LIN {X 0,Y 542.231,Z 590.639,A -85,B 0,C 180,E1 20302.593,E2 20302.593} C_VEL
LIN {X 0,Y 541.639,Z 609.988,A -85,B 0,C 180,E1 20301.85,E2 20301.85} C_VEL
LIN {X 0,Y 540.932,Z 628.979,A -85,B 0,C 180,E1 20300.927,E2 20300.927} C_VEL
LIN {X 0,Y 540.18,Z 647.632,A -85,B 0,C 180,E1 20299.807,E2 20299.807} C_VEL
LIN {X 0,Y 539.393,Z 665.643,A -85,B 0,C 180,E1 20298.495,E2 20298.495} C_VEL
LIN {X 0,Y 538.641,Z 682.161,A -85,B 0,C 180,E1 20297.061,E2 20297.061} C_VEL
LIN {X 0,Y 537.97,Z 697.263,A -85,B 0,C 180,E1 20295.52,E2 20295.52} C_VEL
LIN {X 0,Y 537.346,Z 712.374,A -85,B 0,C 180,E1 20293.707,E2 20293.707} C_VEL
LIN {X 0,Y 536.855,Z 725.652,A -85,B 0,C 180,E1 20291.818,E2 20291.818} C_VEL
LIN {X 0,Y 536.474,Z 737.33,A -85,B 0,C 180,E1 20289.84,E2 20289.84} C_VEL
LIN {X 0,Y 536.224,Z 747.163,A -85,B 0,C 180,E1 20287.841,E2 20287.841} C_VEL
LIN {X 0,Y 536.061,Z 755.619,A -85,B 0,C 180,E1 20285.72,E2 20285.72} C_VEL
LIN {X 0,Y 535.971,Z 762.084,A -85,B 0,C 180,E1 20283.647,E2 20283.647} C_VEL
LIN {X 0,Y 535.926,Z 767.111,A -85,B 0,C 180,E1 20281.493,E2 20281.493} C_VEL
LIN {X 0,Y 535.91,Z 770.431,A -85,B 0,C 180,E1 20279.386,E2 20279.386} C_VEL
LIN {X 0,Y 535.907,Z 772.23,A -85,B 0,C 180,E1 20277.201,E2 20277.201} C_VEL
LIN {X 0,Y 535.911,Z 772.319,A -85,B 0,C 180,E1 20275.058,E2 20275.058} C_VEL
LIN {X 0,Y 535.91,Z 770.761,A -85,B 0,C 180,E1 20272.834,E2 20272.834} C_VEL
LIN {X 0,Y 535.919,Z 767.554,A -85,B 0,C 180,E1 20270.648,E2 20270.648} C_VEL
LIN {X 0,Y 535.954,Z 762.725,A -85,B 0,C 180,E1 20268.491,E2 20268.491} C_VEL
LIN {X 0,Y 536.051,Z 756.221,A -85,B 0,C 180,E1 20266.36,E2 20266.36} C_VEL
LIN {X 0,Y 536.208,Z 747.93,A -85,B 0,C 180,E1 20264.25,E2 20264.25} C_VEL
LIN {X 0,Y 536.444,Z 738.374,A -85,B 0,C 180,E1 20262.269,E2 20262.269} C_VEL
LIN {X 0,Y 536.809,Z 726.982,A -85,B 0,C 180,E1 20260.301,E2 20260.301} C_VEL
LIN {X 0,Y 537.276,Z 714.295,A -85,B 0,C 180,E1 20258.455,E2 20258.455} C_VEL
LIN {X 0,Y 537.858,Z 700.33,A -85,B 0,C 180,E1 20256.727,E2 20256.727} C_VEL
LIN {X 0,Y 538.553,Z 684.434,A -85,B 0,C 180,E1 20255.06,E2 20255.06} C_VEL
LIN {X 0,Y 539.304,Z 667.464,A -85,B 0,C 180,E1 20253.562,E2 20253.562} C_VEL
LIN {X 0,Y 540.049,Z 650.229,A -85,B 0,C 180,E1 20252.282,E2 20252.282} C_VEL
LIN {X 0,Y 540.801,Z 632.241,A -85,B 0,C 180,E1 20251.166,E2 20251.166} C_VEL
LIN {X 0,Y 541.515,Z 613.485,A -85,B 0,C 180,E1 20250.213,E2 20250.213} C_VEL
LIN {X 0,Y 542.159,Z 593.586,A -85,B 0,C 180,E1 20249.413,E2 20249.413} C_VEL
LIN {X 0,Y 542.721,Z 572.923,A -85,B 0,C 180,E1 20248.8,E2 20248.8} C_VEL
LIN {X 0,Y 543.05,Z 552.012,A -85,B 0,C 180,E1 20248.389,E2 20248.389} C_VEL
LIN {X 0,Y 544.939,Z 311.744,A -85,B 0,C 180,E1 20244.932,E2 20244.932} C_VEL
LIN {X 0,Y 542.686,Z 299.098,A -85,B 0,C 180,E1 20244.556,E2 20244.556} C_VEL
LIN {X 0,Y 543.892,Z 265.612,A -85,B 0,C 180,E1 20241.864,E2 20241.864} C_VEL
LIN {X 0,Y 537.565,Z 249.063,A -85,B 0,C 180,E1 20239.932,E2 20239.932} C_VEL
LIN {X 0,Y 536.469,Z 246.09,A -85,B 0,C 180,E1 20239.531,E2 20239.531} C_VEL
LIN {X 0,Y 536.456,Z 245.89,A -85,B 0,C 180,E1 20236.173,E2 20236.173} C_VEL
LIN {X 0,Y 536.46,Z 245.902,A -85,B 0,C 180,E1 20232.763,E2 20232.763} C_VEL
LIN {X 0,Y 536.444,Z 245.913,A -85,B 0,C 180,E1 20229.33,E2 20229.33} C_VEL
LIN {X 0,Y 536.458,Z 245.89,A -85,B 0,C 180,E1 20225.957,E2 20225.957} C_VEL
LIN {X 0,Y 536.466,Z 245.907,A -85,B 0,C 180,E1 20222.471,E2 20222.471} C_VEL
LIN {X 0,Y 536.44,Z 245.909,A -85,B 0,C 180,E1 20219.042,E2 20219.042} C_VEL
LIN {X 0,Y 536.46,Z 245.913,A -85,B 0,C 180,E1 20215.618,E2 20215.618} C_VEL
LIN {X 0,Y 536.461,Z 245.908,A -85,B 0,C 180,E1 20212.181,E2 20212.181} C_VEL
LIN {X 0,Y 536.44,Z 245.91,A -85,B 0,C 180,E1 20208.849,E2 20208.849} C_VEL
LIN {X 0,Y 536.459,Z 245.908,A -85,B 0,C 180,E1 20205.394,E2 20205.394} C_VEL
LIN {X 0,Y 536.46,Z 245.907,A -85,B 0,C 180,E1 20201.958,E2 20201.958} C_VEL
LIN {X 0,Y 536.439,Z 245.91,A -85,B 0,C 180,E1 20198.636,E2 20198.636} C_VEL
LIN {X 0,Y 536.453,Z 245.909,A -85,B 0,C 180,E1 20195.163,E2 20195.163} C_VEL
LIN {X 0,Y 536.46,Z 245.908,A -85,B 0,C 180,E1 20191.707,E2 20191.707} C_VEL
LIN {X 0,Y 536.442,Z 245.909,A -85,B 0,C 180,E1 20188.377,E2 20188.377} C_VEL
LIN {X 0,Y 536.447,Z 245.908,A -85,B 0,C 180,E1 20184.911,E2 20184.911} C_VEL
LIN {X 0,Y 536.462,Z 245.909,A -85,B 0,C 180,E1 20181.54,E2 20181.54} C_VEL
LIN {X 0,Y 536.443,Z 245.906,A -85,B 0,C 180,E1 20178.134,E2 20178.134} C_VEL
LIN {X 0,Y 536.442,Z 245.903,A -85,B 0,C 180,E1 20174.683,E2 20174.683} C_VEL
LIN {X 0,Y 536.46,Z 245.91,A -85,B 0,C 180,E1 20171.285,E2 20171.285} C_VEL
LIN {X 0,Y 536.443,Z 245.901,A -85,B 0,C 180,E1 20167.927,E2 20167.927} C_VEL
LIN {X 0,Y 536.44,Z 245.909,A -85,B 0,C 180,E1 20164.489,E2 20164.489} C_VEL
LIN {X 0,Y 536.461,Z 245.908,A -85,B 0,C 180,E1 20161.067,E2 20161.067} C_VEL
LIN {X 0,Y 536.443,Z 245.901,A -85,B 0,C 180,E1 20157.756,E2 20157.756} C_VEL
LIN {X 0,Y 536.438,Z 245.91,A -85,B 0,C 180,E1 20154.33,E2 20154.33} C_VEL
LIN {X 0,Y 536.462,Z 245.906,A -85,B 0,C 180,E1 20150.992,E2 20150.992} C_VEL
LIN {X 0,Y 536.441,Z 245.9,A -85,B 0,C 180,E1 20147.591,E2 20147.591} C_VEL
LIN {X 0,Y 536.439,Z 245.909,A -85,B 0,C 180,E1 20144.209,E2 20144.209} C_VEL
LIN {X 0,Y 536.463,Z 245.911,A -85,B 0,C 180,E1 20140.85,E2 20140.85} C_VEL
LIN {X 0,Y 536.434,Z 245.91,A -85,B 0,C 180,E1 20137.536,E2 20137.536} C_VEL
LIN {X 0,Y 536.437,Z 245.914,A -85,B 0,C 180,E1 20134.022,E2 20134.022} C_VEL
LIN {X 0,Y 536.464,Z 245.906,A -85,B 0,C 180,E1 20130.647,E2 20130.647} C_VEL
LIN {X 0,Y 536.441,Z 245.908,A -85,B 0,C 180,E1 20127.28,E2 20127.28} C_VEL
LIN {X 0,Y 536.432,Z 245.915,A -85,B 0,C 180,E1 20123.808,E2 20123.808} C_VEL
LIN {X 0,Y 536.465,Z 245.913,A -85,B 0,C 180,E1 20120.496,E2 20120.496} C_VEL
LIN {X 0,Y 536.437,Z 245.908,A -85,B 0,C 180,E1 20117.131,E2 20117.131} C_VEL
LIN {X 0,Y 536.433,Z 245.915,A -85,B 0,C 180,E1 20113.681,E2 20113.681} C_VEL
LIN {X 0,Y 536.457,Z 246.122,A -85,B 0,C 180,E1 20111.282,E2 20111.282} C_VEL
LIN {X 0,Y 537.801,Z 249.457,A -85,B 0,C 180,E1 20110.874,E2 20110.874} C_VEL
LIN {X 0,Y 547.099,Z 269.798,A -85,B 0,C 180,E1 20108.705,E2 20108.705} C_VEL
LIN {X 0,Y 546.078,Z 302.684,A -85,B 0,C 180,E1 20106.578,E2 20106.578} C_VEL
LIN {X 0,Y 548.137,Z 316.155,A -85,B 0,C 180,E1 20106.203,E2 20106.203} C_VEL
LIN {X 0,Y 546.073,Z 534.334,A -85,B 0,C 180,E1 20102.944,E2 20102.944} C_VEL
LIN {X 0,Y 545.342,Z 609.441,A -85,B 0,C 180,E1 20101.809,E2 20101.809} C_VEL
LIN {X 0,Y 544.74,Z 631.09,A -85,B 0,C 180,E1 20101.285,E2 20101.285} C_VEL
LIN {X 0,Y 544.045,Z 653.257,A -85,B 0,C 180,E1 20100.54,E2 20100.54} C_VEL
LIN {X 0,Y 543.252,Z 673.418,A -85,B 0,C 180,E1 20099.674,E2 20099.674} C_VEL
LIN {X 0,Y 542.321,Z 693.777,A -85,B 0,C 180,E1 20098.581,E2 20098.581} C_VEL
LIN {X 0,Y 541.316,Z 714.156,A -85,B 0,C 180,E1 20097.262,E2 20097.262} C_VEL
LIN {X 0,Y 540.361,Z 732.791,A -85,B 0,C 180,E1 20095.832,E2 20095.832} C_VEL
LIN {X 0,Y 539.448,Z 750.618,A -85,B 0,C 180,E1 20094.229,E2 20094.229} C_VEL
LIN {X 0,Y 538.586,Z 767.204,A -85,B 0,C 180,E1 20092.483,E2 20092.483} C_VEL
LIN {X 0,Y 537.832,Z 782.883,A -85,B 0,C 180,E1 20090.569,E2 20090.569} C_VEL
LIN {X 0,Y 537.224,Z 797.055,A -85,B 0,C 180,E1 20088.556,E2 20088.556} C_VEL
LIN {X 0,Y 536.748,Z 809.739,A -85,B 0,C 180,E1 20086.447,E2 20086.447} C_VEL
LIN {X 0,Y 536.402,Z 820.339,A -85,B 0,C 180,E1 20084.353,E2 20084.353} C_VEL
LIN {X 0,Y 536.157,Z 830.075,A -85,B 0,C 180,E1 20082.055,E2 20082.055} C_VEL
LIN {X 0,Y 536.017,Z 837.94,A -85,B 0,C 180,E1 20079.772,E2 20079.772} C_VEL
LIN {X 0,Y 535.945,Z 843.91,A -85,B 0,C 180,E1 20077.503,E2 20077.503} C_VEL
LIN {X 0,Y 535.924,Z 848.465,A -85,B 0,C 180,E1 20075.137,E2 20075.137} C_VEL
LIN {X 0,Y 535.912,Z 851.236,A -85,B 0,C 180,E1 20072.886,E2 20072.886} C_VEL
LIN {X 0,Y 535.898,Z 852.373,A -85,B 0,C 180,E1 20070.64,E2 20070.64} C_VEL
LIN {X 0,Y 535.9,Z 852.015,A -85,B 0,C 180,E1 20068.288,E2 20068.288} C_VEL
LIN {X 0,Y 535.908,Z 850.219,A -85,B 0,C 180,E1 20066.148,E2 20066.148} C_VEL
LIN {X 0,Y 535.926,Z 846.601,A -85,B 0,C 180,E1 20063.787,E2 20063.787} C_VEL
LIN {X 0,Y 535.969,Z 841.58,A -85,B 0,C 180,E1 20061.524,E2 20061.524} C_VEL
LIN {X 0,Y 536.06,Z 835.109,A -85,B 0,C 180,E1 20059.358,E2 20059.358} C_VEL
LIN {X 0,Y 536.233,Z 826.595,A -85,B 0,C 180,E1 20057.07,E2 20057.07} C_VEL
LIN {X 0,Y 536.512,Z 816.68,A -85,B 0,C 180,E1 20054.875,E2 20054.875} C_VEL
LIN {X 0,Y 536.895,Z 805.267,A -85,B 0,C 180,E1 20052.775,E2 20052.775} C_VEL
LIN {X 0,Y 537.446,Z 791.783,A -85,B 0,C 180,E1 20050.661,E2 20050.661} C_VEL
LIN {X 0,Y 538.093,Z 777.646,A -85,B 0,C 180,E1 20048.755,E2 20048.755} C_VEL
LIN {X 0,Y 538.888,Z 761.61,A -85,B 0,C 180,E1 20046.894,E2 20046.894} C_VEL
LIN {X 0,Y 539.741,Z 744.45,A -85,B 0,C 180,E1 20045.191,E2 20045.191} C_VEL
LIN {X 0,Y 540.728,Z 725.653,A -85,B 0,C 180,E1 20043.594,E2 20043.594} C_VEL
LIN {X 0,Y 541.712,Z 706.636,A -85,B 0,C 180,E1 20042.221,E2 20042.221} C_VEL
LIN {X 0,Y 542.581,Z 687.942,A -85,B 0,C 180,E1 20041.083,E2 20041.083} C_VEL
LIN {X 0,Y 543.485,Z 667.482,A -85,B 0,C 180,E1 20040.055,E2 20040.055} C_VEL
LIN {X 0,Y 544.282,Z 646.805,A -85,B 0,C 180,E1 20039.216,E2 20039.216} C_VEL
LIN {X 0,Y 544.911,Z 626.046,A -85,B 0,C 180,E1 20038.576,E2 20038.576} C_VEL
LIN {X 0,Y 545.407,Z 603.72,A -85,B 0,C 180,E1 20038.091,E2 20038.091} C_VEL
LIN {X 0,Y 547.479,Z 382.783,A -85,B 0,C 180,E1 20034.802,E2 20034.802} C_VEL
LIN {X 0,Y 547.957,Z 313.802,A -85,B 0,C 180,E1 20033.746,E2 20033.746} C_VEL
LIN {X 0,Y 545.988,Z 301.611,A -85,B 0,C 180,E1 20033.377,E2 20033.377} C_VEL
LIN {X 0,Y 547.099,Z 269.797,A -85,B 0,C 180,E1 20031.295,E2 20031.295} C_VEL
LIN {X 0,Y 536.506,Z 246.372,A -85,B 0,C 180,E1 20028.795,E2 20028.795} C_VEL
LIN {X 0,Y 536.433,Z 245.902,A -85,B 0,C 180,E1 20028.529,E2 20028.529} C_VEL
LIN {X 0,Y 536.452,Z 245.911,A -85,B 0,C 180,E1 20025.057,E2 20025.057} C_VEL
LIN {X 0,Y 536.46,Z 245.913,A -85,B 0,C 180,E1 20021.635,E2 20021.635} C_VEL
LIN {X 0,Y 536.451,Z 245.913,A -85,B 0,C 180,E1 20018.229,E2 20018.229} C_VEL
LIN {X 0,Y 536.448,Z 245.911,A -85,B 0,C 180,E1 20014.718,E2 20014.718} C_VEL
LIN {X 0,Y 536.455,Z 245.909,A -85,B 0,C 180,E1 20011.333,E2 20011.333} C_VEL
LIN {X 0,Y 536.463,Z 245.915,A -85,B 0,C 180,E1 20007.893,E2 20007.893} C_VEL
LIN {X 0,Y 536.452,Z 245.911,A -85,B 0,C 180,E1 20004.443,E2 20004.443} C_VEL
LIN {X 0,Y 536.453,Z 245.906,A -85,B 0,C 180,E1 20001.084,E2 20001.084} C_VEL
LIN {X 0,Y 536.445,Z 245.91,A -85,B 0,C 180,E1 19997.575,E2 19997.575} C_VEL
LIN {X 0,Y 536.459,Z 245.91,A -85,B 0,C 180,E1 19994.243,E2 19994.243} C_VEL
LIN {X 0,Y 536.455,Z 245.903,A -85,B 0,C 180,E1 19990.813,E2 19990.813} C_VEL
LIN {X 0,Y 536.433,Z 245.912,A -85,B 0,C 180,E1 19987.39,E2 19987.39} C_VEL
LIN {X 0,Y 536.462,Z 245.909,A -85,B 0,C 180,E1 19984.062,E2 19984.062} C_VEL
LIN {X 0,Y 536.454,Z 245.907,A -85,B 0,C 180,E1 19980.642,E2 19980.642} C_VEL
LIN {X 0,Y 536.422,Z 245.913,A -85,B 0,C 180,E1 19977.223,E2 19977.223} C_VEL
LIN {X 0,Y 536.461,Z 245.914,A -85,B 0,C 180,E1 19973.903,E2 19973.903} C_VEL
LIN {X 0,Y 536.442,Z 245.911,A -85,B 0,C 180,E1 19970.561,E2 19970.561} C_VEL
LIN {X 0,Y 536.412,Z 245.915,A -85,B 0,C 180,E1 19967.186,E2 19967.186} C_VEL
LIN {X 0,Y 536.458,Z 245.913,A -85,B 0,C 180,E1 19963.878,E2 19963.878} C_VEL
LIN {X 0,Y 536.421,Z 245.915,A -85,B 0,C 180,E1 19960.59,E2 19960.59} C_VEL
LIN {X 0,Y 536.401,Z 245.907,A -85,B 0,C 180,E1 19957.189,E2 19957.189} C_VEL
LIN {X 0,Y 536.46,Z 245.902,A -85,B 0,C 180,E1 19953.907,E2 19953.907} C_VEL
LIN {X 0,Y 536.435,Z 246.067,A -85,B 0,C 180,E1 19952.469,E2 19952.469} C_VEL
LIN {X 0,Y 537.144,Z 248.318,A -85,B 0,C 180,E1 19952.148,E2 19952.148} C_VEL
LIN {X 0,Y 543.179,Z 263.493,A -85,B 0,C 180,E1 19950.321,E2 19950.321} C_VEL
LIN {X 0,Y 544.043,Z 266.321,A -85,B 0,C 180,E1 19950.009,E2 19950.009} C_VEL
LIN {X 0,Y 542.886,Z 293.11,A -85,B 0,C 180,E1 19947.831,E2 19947.831} C_VEL
LIN {X 0,Y 542.449,Z 298.495,A -85,B 0,C 180,E1 19947.531,E2 19947.531} C_VEL
LIN {X 0,Y 541.467,Z 305.679,A -85,B 0,C 180,E1 19947.356,E2 19947.356} C_VEL
LIN {X 0,Y 538.242,Z 325.089,A -85,B 0,C 180,E1 19947.245,E2 19947.245} C_VEL
LIN {X 0,Y 538.106,Z 328.159,A -85,B 0,C 180,E1 19947.206,E2 19947.206} C_VEL
LIN {X 0,Y 536.108,Z 536.437,A -85,B 0,C 180,E1 19944.146,E2 19944.146} C_VEL
LIN {X 0,Y 535.736,Z 564.945,A -85,B 0,C 180,E1 19943.681,E2 19943.681} C_VEL
LIN {X 0,Y 535.249,Z 585.172,A -85,B 0,C 180,E1 19943.158,E2 19943.158} C_VEL
LIN {X 0,Y 534.567,Z 605.412,A -85,B 0,C 180,E1 19942.43,E2 19942.43} C_VEL
LIN {X 0,Y 533.801,Z 624.508,A -85,B 0,C 180,E1 19941.533,E2 19941.533} C_VEL
LIN {X 0,Y 532.944,Z 643.109,A -85,B 0,C 180,E1 19940.452,E2 19940.452} C_VEL
LIN {X 0,Y 532.051,Z 661.433,A -85,B 0,C 180,E1 19939.16,E2 19939.16} C_VEL
LIN {X 0,Y 531.194,Z 678.609,A -85,B 0,C 180,E1 19937.71,E2 19937.71} C_VEL
LIN {X 0,Y 530.414,Z 694.38,A -85,B 0,C 180,E1 19936.138,E2 19936.138} C_VEL
LIN {X 0,Y 529.714,Z 709.19,A -85,B 0,C 180,E1 19934.399,E2 19934.399} C_VEL
LIN {X 0,Y 529.128,Z 722.654,A -85,B 0,C 180,E1 19932.529,E2 19932.529} C_VEL
LIN {X 0,Y 528.666,Z 734.421,A -85,B 0,C 180,E1 19930.588,E2 19930.588} C_VEL
LIN {X 0,Y 528.347,Z 744.525,A -85,B 0,C 180,E1 19928.598,E2 19928.598} C_VEL
LIN {X 0,Y 528.117,Z 753.561,A -85,B 0,C 180,E1 19926.428,E2 19926.428} C_VEL
LIN {X 0,Y 527.992,Z 760.468,A -85,B 0,C 180,E1 19924.348,E2 19924.348} C_VEL
LIN {X 0,Y 527.934,Z 766.005,A -85,B 0,C 180,E1 19922.154,E2 19922.154} C_VEL
LIN {X 0,Y 527.916,Z 769.705,A -85,B 0,C 180,E1 19920.002,E2 19920.002} C_VEL
LIN {X 0,Y 527.912,Z 771.893,A -85,B 0,C 180,E1 19917.771,E2 19917.771} C_VEL
LIN {X 0,Y 527.909,Z 772.406,A -85,B 0,C 180,E1 19915.465,E2 19915.465} C_VEL
LIN {X 0,Y 527.916,Z 771.277,A -85,B 0,C 180,E1 19913.286,E2 19913.286} C_VEL
LIN {X 0,Y 527.927,Z 768.509,A -85,B 0,C 180,E1 19911.092,E2 19911.092} C_VEL
LIN {X 0,Y 527.95,Z 764.012,A -85,B 0,C 180,E1 19908.897,E2 19908.897} C_VEL
LIN {X 0,Y 528.031,Z 757.881,A -85,B 0,C 180,E1 19906.729,E2 19906.729} C_VEL
LIN {X 0,Y 528.198,Z 750.062,A -85,B 0,C 180,E1 19904.583,E2 19904.583} C_VEL
LIN {X 0,Y 528.461,Z 740.712,A -85,B 0,C 180,E1 19902.512,E2 19902.512} C_VEL
LIN {X 0,Y 528.856,Z 729.463,A -85,B 0,C 180,E1 19900.458,E2 19900.458} C_VEL
LIN {X 0,Y 529.389,Z 716.399,A -85,B 0,C 180,E1 19898.473,E2 19898.473} C_VEL
LIN {X 0,Y 530.06,Z 701.803,A -85,B 0,C 180,E1 19896.608,E2 19896.608} C_VEL
LIN {X 0,Y 530.795,Z 686.667,A -85,B 0,C 180,E1 19894.972,E2 19894.972} C_VEL
LIN {X 0,Y 531.616,Z 670.115,A -85,B 0,C 180,E1 19893.452,E2 19893.452} C_VEL
LIN {X 0,Y 532.526,Z 651.863,A -85,B 0,C 180,E1 19892.046,E2 19892.046} C_VEL
LIN {X 0,Y 533.404,Z 633.281,A -85,B 0,C 180,E1 19890.86,E2 19890.86} C_VEL
LIN {X 0,Y 534.203,Z 614.771,A -85,B 0,C 180,E1 19889.894,E2 19889.894} C_VEL
LIN {X 0,Y 534.94,Z 594.645,A -85,B 0,C 180,E1 19889.064,E2 19889.064} C_VEL
LIN {X 0,Y 535.55,Z 574.091,A -85,B 0,C 180,E1 19888.44,E2 19888.44} C_VEL
LIN {X 0,Y 535.932,Z 553.561,A -85,B 0,C 180,E1 19888.018,E2 19888.018} C_VEL
LIN {X 0,Y 538.226,Z 313.309,A -85,B 0,C 180,E1 19884.491,E2 19884.491} C_VEL
LIN {X 0,Y 535.703,Z 298.99,A -85,B 0,C 180,E1 19884.05,E2 19884.05} C_VEL
LIN {X 0,Y 536.908,Z 268.83,A -85,B 0,C 180,E1 19881.595,E2 19881.595} C_VEL
LIN {X 0,Y 530.553,Z 252.496,A -85,B 0,C 180,E1 19879.643,E2 19879.643} C_VEL
LIN {X 0,Y 528.552,Z 247.144,A -85,B 0,C 180,E1 19878.959,E2 19878.959} C_VEL
LIN {X 0,Y 528.505,Z 246.883,A -85,B 0,C 180,E1 19875.54,E2 19875.54} C_VEL
LIN {X 0,Y 528.517,Z 246.88,A -85,B 0,C 180,E1 19872.155,E2 19872.155} C_VEL
LIN {X 0,Y 528.525,Z 246.897,A -85,B 0,C 180,E1 19868.703,E2 19868.703} C_VEL
LIN {X 0,Y 528.501,Z 246.89,A -85,B 0,C 180,E1 19865.24,E2 19865.24} C_VEL
LIN {X 0,Y 528.523,Z 246.898,A -85,B 0,C 180,E1 19861.83,E2 19861.83} C_VEL
LIN {X 0,Y 528.525,Z 246.894,A -85,B 0,C 180,E1 19858.351,E2 19858.351} C_VEL
LIN {X 0,Y 528.502,Z 246.894,A -85,B 0,C 180,E1 19854.893,E2 19854.893} C_VEL
LIN {X 0,Y 528.524,Z 246.899,A -85,B 0,C 180,E1 19851.51,E2 19851.51} C_VEL
LIN {X 0,Y 528.518,Z 246.898,A -85,B 0,C 180,E1 19848.027,E2 19848.027} C_VEL
LIN {X 0,Y 528.507,Z 246.896,A -85,B 0,C 180,E1 19844.576,E2 19844.576} C_VEL
LIN {X 0,Y 528.504,Z 246.895,A -85,B 0,C 180,E1 19841.03,E2 19841.03} C_VEL
LIN {X 0,Y 528.521,Z 246.9,A -85,B 0,C 180,E1 19837.664,E2 19837.664} C_VEL
LIN {X 0,Y 528.518,Z 246.894,A -85,B 0,C 180,E1 19834.183,E2 19834.183} C_VEL
LIN {X 0,Y 528.5,Z 246.893,A -85,B 0,C 180,E1 19830.716,E2 19830.716} C_VEL
LIN {X 0,Y 528.525,Z 246.902,A -85,B 0,C 180,E1 19827.367,E2 19827.367} C_VEL
LIN {X 0,Y 528.522,Z 246.892,A -85,B 0,C 180,E1 19823.88,E2 19823.88} C_VEL
LIN {X 0,Y 528.497,Z 246.892,A -85,B 0,C 180,E1 19820.486,E2 19820.486} C_VEL
LIN {X 0,Y 528.522,Z 246.903,A -85,B 0,C 180,E1 19817.05,E2 19817.05} C_VEL
LIN {X 0,Y 528.523,Z 246.886,A -85,B 0,C 180,E1 19813.566,E2 19813.566} C_VEL
LIN {X 0,Y 528.499,Z 246.896,A -85,B 0,C 180,E1 19810.133,E2 19810.133} C_VEL
LIN {X 0,Y 528.507,Z 246.903,A -85,B 0,C 180,E1 19806.626,E2 19806.626} C_VEL
LIN {X 0,Y 528.522,Z 246.895,A -85,B 0,C 180,E1 19803.253,E2 19803.253} C_VEL
LIN {X 0,Y 528.5,Z 246.898,A -85,B 0,C 180,E1 19799.891,E2 19799.891} C_VEL
LIN {X 0,Y 528.503,Z 246.901,A -85,B 0,C 180,E1 19796.42,E2 19796.42} C_VEL
LIN {X 0,Y 528.524,Z 246.897,A -85,B 0,C 180,E1 19793.045,E2 19793.045} C_VEL
LIN {X 0,Y 528.504,Z 246.897,A -85,B 0,C 180,E1 19789.645,E2 19789.645} C_VEL
LIN {X 0,Y 528.499,Z 246.902,A -85,B 0,C 180,E1 19786.209,E2 19786.209} C_VEL
LIN {X 0,Y 528.524,Z 246.893,A -85,B 0,C 180,E1 19782.809,E2 19782.809} C_VEL
LIN {X 0,Y 528.507,Z 246.894,A -85,B 0,C 180,E1 19779.397,E2 19779.397} C_VEL
LIN {X 0,Y 528.495,Z 246.899,A -85,B 0,C 180,E1 19775.998,E2 19775.998} C_VEL
LIN {X 0,Y 528.526,Z 246.902,A -85,B 0,C 180,E1 19772.631,E2 19772.631} C_VEL
LIN {X 0,Y 528.512,Z 246.899,A -85,B 0,C 180,E1 19769.156,E2 19769.156} C_VEL
LIN {X 0,Y 528.491,Z 246.899,A -85,B 0,C 180,E1 19765.681,E2 19765.681} C_VEL
LIN {X 0,Y 528.523,Z 246.897,A -85,B 0,C 180,E1 19762.255,E2 19762.255} C_VEL
LIN {X 0,Y 528.526,Z 246.896,A -85,B 0,C 180,E1 19758.826,E2 19758.826} C_VEL
LIN {X 0,Y 528.487,Z 246.88,A -85,B 0,C 180,E1 19755.42,E2 19755.42} C_VEL
LIN {X 0,Y 528.523,Z 246.975,A -85,B 0,C 180,E1 19751.956,E2 19751.956} C_VEL
LIN {X 0,Y 528.778,Z 248.203,A -85,B 0,C 180,E1 19751.759,E2 19751.759} C_VEL
LIN {X 0,Y 540.318,Z 273.235,A -85,B 0,C 180,E1 19749.015,E2 19749.015} C_VEL
LIN {X 0,Y 539.401,Z 302.735,A -85,B 0,C 180,E1 19747.105,E2 19747.105} C_VEL
LIN {X 0,Y 541.667,Z 317.551,A -85,B 0,C 180,E1 19746.682,E2 19746.682} C_VEL
LIN {X 0,Y 539.35,Z 535.509,A -85,B 0,C 180,E1 19743.389,E2 19743.389} C_VEL
LIN {X 0,Y 538.541,Z 609.44,A -85,B 0,C 180,E1 19742.259,E2 19742.259} C_VEL
LIN {X 0,Y 537.874,Z 631.088,A -85,B 0,C 180,E1 19741.731,E2 19741.731} C_VEL
LIN {X 0,Y 537.102,Z 653.254,A -85,B 0,C 180,E1 19740.977,E2 19740.977} C_VEL
LIN {X 0,Y 536.194,Z 673.693,A -85,B 0,C 180,E1 19740.09,E2 19740.09} C_VEL
LIN {X 0,Y 535.176,Z 693.681,A -85,B 0,C 180,E1 19739.005,E2 19739.005} C_VEL
LIN {X 0,Y 534.037,Z 714.152,A -85,B 0,C 180,E1 19737.665,E2 19737.665} C_VEL
LIN {X 0,Y 532.933,Z 733.456,A -85,B 0,C 180,E1 19736.159,E2 19736.159} C_VEL
LIN {X 0,Y 531.902,Z 751.374,A -85,B 0,C 180,E1 19734.52,E2 19734.52} C_VEL
LIN {X 0,Y 530.914,Z 768.216,A -85,B 0,C 180,E1 19732.709,E2 19732.709} C_VEL
LIN {X 0,Y 530.066,Z 783.729,A -85,B 0,C 180,E1 19730.769,E2 19730.769} C_VEL
LIN {X 0,Y 529.384,Z 797.763,A -85,B 0,C 180,E1 19728.727,E2 19728.727} C_VEL
LIN {X 0,Y 528.852,Z 810.357,A -85,B 0,C 180,E1 19726.586,E2 19726.586} C_VEL
LIN {X 0,Y 528.448,Z 821.299,A -85,B 0,C 180,E1 19724.364,E2 19724.364} C_VEL
LIN {X 0,Y 528.186,Z 830.483,A -85,B 0,C 180,E1 19722.128,E2 19722.128} C_VEL
LIN {X 0,Y 528.035,Z 837.94,A -85,B 0,C 180,E1 19719.921,E2 19719.921} C_VEL
LIN {X 0,Y 527.954,Z 843.91,A -85,B 0,C 180,E1 19717.617,E2 19717.617} C_VEL
LIN {X 0,Y 527.925,Z 848.465,A -85,B 0,C 180,E1 19715.215,E2 19715.215} C_VEL
LIN {X 0,Y 527.912,Z 851.236,A -85,B 0,C 180,E1 19712.93,E2 19712.93} C_VEL
LIN {X 0,Y 527.898,Z 852.373,A -85,B 0,C 180,E1 19710.65,E2 19710.65} C_VEL
LIN {X 0,Y 527.901,Z 852.015,A -85,B 0,C 180,E1 19708.262,E2 19708.262} C_VEL
LIN {X 0,Y 527.909,Z 850.218,A -85,B 0,C 180,E1 19706.089,E2 19706.089} C_VEL
LIN {X 0,Y 527.926,Z 846.601,A -85,B 0,C 180,E1 19703.692,E2 19703.692} C_VEL
LIN {X 0,Y 527.974,Z 841.58,A -85,B 0,C 180,E1 19701.395,E2 19701.395} C_VEL
LIN {X 0,Y 528.082,Z 835.109,A -85,B 0,C 180,E1 19699.195,E2 19699.195} C_VEL
LIN {X 0,Y 528.285,Z 826.594,A -85,B 0,C 180,E1 19696.872,E2 19696.872} C_VEL
LIN {X 0,Y 528.609,Z 816.681,A -85,B 0,C 180,E1 19694.643,E2 19694.643} C_VEL
LIN {X 0,Y 529.045,Z 805.268,A -85,B 0,C 180,E1 19692.511,E2 19692.511} C_VEL
LIN {X 0,Y 529.666,Z 791.782,A -85,B 0,C 180,E1 19690.365,E2 19690.365} C_VEL
LIN {X 0,Y 530.403,Z 777.645,A -85,B 0,C 180,E1 19688.432,E2 19688.432} C_VEL
LIN {X 0,Y 531.29,Z 761.845,A -85,B 0,C 180,E1 19686.571,E2 19686.571} C_VEL
LIN {X 0,Y 532.241,Z 745.048,A -85,B 0,C 180,E1 19684.876,E2 19684.876} C_VEL
LIN {X 0,Y 533.337,Z 726.385,A -85,B 0,C 180,E1 19683.26,E2 19683.26} C_VEL
LIN {X 0,Y 534.445,Z 707.529,A -85,B 0,C 180,E1 19681.871,E2 19681.871} C_VEL
LIN {X 0,Y 535.475,Z 687.72,A -85,B 0,C 180,E1 19680.649,E2 19680.649} C_VEL
LIN {X 0,Y 536.49,Z 667.145,A -85,B 0,C 180,E1 19679.608,E2 19679.608} C_VEL
LIN {X 0,Y 537.367,Z 646.377,A -85,B 0,C 180,E1 19678.761,E2 19678.761} C_VEL
LIN {X 0,Y 538.08,Z 625.648,A -85,B 0,C 180,E1 19678.119,E2 19678.119} C_VEL
LIN {X 0,Y 538.616,Z 603.419,A -85,B 0,C 180,E1 19677.635,E2 19677.635} C_VEL
LIN {X 0,Y 540.921,Z 384.819,A -85,B 0,C 180,E1 19674.343,E2 19674.343} C_VEL
LIN {X 0,Y 541.495,Z 315.285,A -85,B 0,C 180,E1 19673.267,E2 19673.267} C_VEL
LIN {X 0,Y 539.307,Z 301.906,A -85,B 0,C 180,E1 19672.864,E2 19672.864} C_VEL
LIN {X 0,Y 540.153,Z 272.812,A -85,B 0,C 180,E1 19670.952,E2 19670.952} C_VEL
LIN {X 0,Y 528.584,Z 247.376,A -85,B 0,C 180,E1 19668.184,E2 19668.184} C_VEL
LIN {X 0,Y 528.524,Z 246.893,A -85,B 0,C 180,E1 19667.867,E2 19667.867} C_VEL
LIN {X 0,Y 528.502,Z 246.904,A -85,B 0,C 180,E1 19664.427,E2 19664.427} C_VEL
LIN {X 0,Y 528.51,Z 246.901,A -85,B 0,C 180,E1 19660.888,E2 19660.888} C_VEL
LIN {X 0,Y 528.519,Z 246.902,A -85,B 0,C 180,E1 19657.529,E2 19657.529} C_VEL
LIN {X 0,Y 528.519,Z 246.9,A -85,B 0,C 180,E1 19654.042,E2 19654.042} C_VEL
LIN {X 0,Y 528.509,Z 246.899,A -85,B 0,C 180,E1 19650.592,E2 19650.592} C_VEL
LIN {X 0,Y 528.516,Z 246.897,A -85,B 0,C 180,E1 19647.231,E2 19647.231} C_VEL
LIN {X 0,Y 528.514,Z 246.899,A -85,B 0,C 180,E1 19643.701,E2 19643.701} C_VEL
LIN {X 0,Y 528.518,Z 246.897,A -85,B 0,C 180,E1 19640.371,E2 19640.371} C_VEL
LIN {X 0,Y 528.517,Z 246.894,A -85,B 0,C 180,E1 19636.939,E2 19636.939} C_VEL
LIN {X 0,Y 528.501,Z 246.902,A -85,B 0,C 180,E1 19633.457,E2 19633.457} C_VEL
LIN {X 0,Y 528.523,Z 246.899,A -85,B 0,C 180,E1 19630.024,E2 19630.024} C_VEL
LIN {X 0,Y 528.526,Z 246.896,A -85,B 0,C 180,E1 19626.518,E2 19626.518} C_VEL
LIN {X 0,Y 528.49,Z 246.901,A -85,B 0,C 180,E1 19623.146,E2 19623.146} C_VEL
LIN {X 0,Y 528.504,Z 246.902,A -85,B 0,C 180,E1 19619.676,E2 19619.676} C_VEL
LIN {X 0,Y 528.526,Z 246.9,A -85,B 0,C 180,E1 19616.313,E2 19616.313} C_VEL
LIN {X 0,Y 528.481,Z 246.898,A -85,B 0,C 180,E1 19612.937,E2 19612.937} C_VEL
LIN {X 0,Y 528.483,Z 246.905,A -85,B 0,C 180,E1 19609.426,E2 19609.426} C_VEL
LIN {X 0,Y 528.531,Z 246.901,A -85,B 0,C 180,E1 19606.045,E2 19606.045} C_VEL
LIN {X 0,Y 528.477,Z 246.904,A -85,B 0,C 180,E1 19602.721,E2 19602.721} C_VEL
LIN {X 0,Y 528.47,Z 246.907,A -85,B 0,C 180,E1 19599.281,E2 19599.281} C_VEL
LIN {X 0,Y 528.521,Z 246.899,A -85,B 0,C 180,E1 19596.001,E2 19596.001} C_VEL
LIN {X 0,Y 528.468,Z 246.982,A -85,B 0,C 180,E1 19593.117,E2 19593.117} C_VEL
LIN {X 0,Y 528.757,Z 248.299,A -85,B 0,C 180,E1 19592.89,E2 19592.89} C_VEL
LIN {X 0,Y 534.532,Z 262.196,A -85,B 0,C 180,E1 19591.146,E2 19591.146} C_VEL
LIN {X 0,Y 537.093,Z 269.901,A -85,B 0,C 180,E1 19590.258,E2 19590.258} C_VEL
LIN {X 0,Y 535.82,Z 299.702,A -85,B 0,C 180,E1 19587.842,E2 19587.842} C_VEL
LIN {X 0,Y 538.278,Z 314.203,A -85,B 0,C 180,E1 19587.416,E2 19587.416} C_VEL
LIN {X 0,Y 538.106,Z 328.159,A -85,B 0,C 180,E1 19587.206,E2 19587.206} C_VEL
LIN {X 0,Y 537.196,Z 335.853,A -85,B 0,C 180,E1 19587.15,E2 19587.15} C_VEL
LIN {X 0,Y 531.753,Z 356.385,A -85,B 0,C 180,E1 19587.218,E2 19587.218} C_VEL
LIN {X 0,Y 531.049,Z 362.988,A -85,B 0,C 180,E1 19587.164,E2 19587.164} C_VEL
LIN {X 0,Y 528.774,Z 561.36,A -85,B 0,C 180,E1 19584.166,E2 19584.166} C_VEL
LIN {X 0,Y 528.177,Z 583.04,A -85,B 0,C 180,E1 19583.625,E2 19583.625} C_VEL
LIN {X 0,Y 527.462,Z 602.612,A -85,B 0,C 180,E1 19582.931,E2 19582.931} C_VEL
LIN {X 0,Y 526.615,Z 622.066,A -85,B 0,C 180,E1 19582.038,E2 19582.038} C_VEL
LIN {X 0,Y 525.617,Z 641.737,A -85,B 0,C 180,E1 19580.908,E2 19580.908} C_VEL
LIN {X 0,Y 524.651,Z 660.103,A -85,B 0,C 180,E1 19579.614,E2 19579.614} C_VEL
LIN {X 0,Y 523.736,Z 676.69,A -85,B 0,C 180,E1 19578.222,E2 19578.222} C_VEL
LIN {X 0,Y 522.832,Z 692.906,A -85,B 0,C 180,E1 19576.612,E2 19576.612} C_VEL
LIN {X 0,Y 522.002,Z 708.115,A -85,B 0,C 180,E1 19574.821,E2 19574.821} C_VEL
LIN {X 0,Y 521.321,Z 721.798,A -85,B 0,C 180,E1 19572.912,E2 19572.912} C_VEL
LIN {X 0,Y 520.815,Z 733.253,A -85,B 0,C 180,E1 19571.023,E2 19571.023} C_VEL
LIN {X 0,Y 520.421,Z 743.97,A -85,B 0,C 180,E1 19568.915,E2 19568.915} C_VEL
LIN {X 0,Y 520.179,Z 752.619,A -85,B 0,C 180,E1 19566.85,E2 19566.85} C_VEL
LIN {X 0,Y 520.023,Z 759.884,A -85,B 0,C 180,E1 19564.69,E2 19564.69} C_VEL
LIN {X 0,Y 519.943,Z 765.628,A -85,B 0,C 180,E1 19562.417,E2 19562.417} C_VEL
LIN {X 0,Y 519.916,Z 769.429,A -85,B 0,C 180,E1 19560.256,E2 19560.256} C_VEL
LIN {X 0,Y 519.914,Z 771.776,A -85,B 0,C 180,E1 19557.986,E2 19557.986} C_VEL
LIN {X 0,Y 519.908,Z 772.468,A -85,B 0,C 180,E1 19555.763,E2 19555.763} C_VEL
LIN {X 0,Y 519.908,Z 771.565,A -85,B 0,C 180,E1 19553.58,E2 19553.58} C_VEL
LIN {X 0,Y 519.917,Z 769.109,A -85,B 0,C 180,E1 19551.433,E2 19551.433} C_VEL
LIN {X 0,Y 519.953,Z 764.953,A -85,B 0,C 180,E1 19549.199,E2 19549.199} C_VEL
LIN {X 0,Y 520.034,Z 759.175,A -85,B 0,C 180,E1 19546.994,E2 19546.994} C_VEL
LIN {X 0,Y 520.202,Z 751.713,A -85,B 0,C 180,E1 19544.812,E2 19544.812} C_VEL
LIN {X 0,Y 520.486,Z 742.247,A -85,B 0,C 180,E1 19542.62,E2 19542.62} C_VEL
LIN {X 0,Y 520.879,Z 731.75,A -85,B 0,C 180,E1 19540.62,E2 19540.62} C_VEL
LIN {X 0,Y 521.402,Z 719.88,A -85,B 0,C 180,E1 19538.715,E2 19538.715} C_VEL
LIN {X 0,Y 522.108,Z 705.938,A -85,B 0,C 180,E1 19536.82,E2 19536.82} C_VEL
LIN {X 0,Y 522.893,Z 691.571,A -85,B 0,C 180,E1 19535.157,E2 19535.157} C_VEL
LIN {X 0,Y 523.818,Z 675.288,A -85,B 0,C 180,E1 19533.558,E2 19533.558} C_VEL
LIN {X 0,Y 524.829,Z 657.274,A -85,B 0,C 180,E1 19532.076,E2 19532.076} C_VEL
LIN {X 0,Y 525.784,Z 638.846,A -85,B 0,C 180,E1 19530.818,E2 19530.818} C_VEL
LIN {X 0,Y 526.689,Z 620.345,A -85,B 0,C 180,E1 19529.784,E2 19529.784} C_VEL
LIN {X 0,Y 527.546,Z 600.295,A -85,B 0,C 180,E1 19528.888,E2 19528.888} C_VEL
LIN {X 0,Y 528.227,Z 580.312,A -85,B 0,C 180,E1 19528.208,E2 19528.208} C_VEL
LIN {X 0,Y 528.795,Z 559.706,A -85,B 0,C 180,E1 19527.715,E2 19527.715} C_VEL
LIN {X 0,Y 531.551,Z 314.557,A -85,B 0,C 180,E1 19524.029,E2 19524.029} C_VEL
LIN {X 0,Y 528.753,Z 299.04,A -85,B 0,C 180,E1 19523.541,E2 19523.541} C_VEL
LIN {X 0,Y 529.914,Z 272.066,A -85,B 0,C 180,E1 19521.319,E2 19521.319} C_VEL
LIN {X 0,Y 523.182,Z 254.633,A -85,B 0,C 180,E1 19519.198,E2 19519.198} C_VEL
LIN {X 0,Y 520.616,Z 248.152,A -85,B 0,C 180,E1 19518.342,E2 19518.342} C_VEL
LIN {X 0,Y 520.567,Z 247.875,A -85,B 0,C 180,E1 19515.201,E2 19515.201} C_VEL
LIN {X 0,Y 520.577,Z 247.865,A -85,B 0,C 180,E1 19511.757,E2 19511.757} C_VEL
LIN {X 0,Y 520.579,Z 247.887,A -85,B 0,C 180,E1 19508.243,E2 19508.243} C_VEL
LIN {X 0,Y 520.575,Z 247.881,A -85,B 0,C 180,E1 19504.763,E2 19504.763} C_VEL
LIN {X 0,Y 520.567,Z 247.888,A -85,B 0,C 180,E1 19501.305,E2 19501.305} C_VEL
LIN {X 0,Y 520.581,Z 247.884,A -85,B 0,C 180,E1 19497.86,E2 19497.86} C_VEL
LIN {X 0,Y 520.583,Z 247.88,A -85,B 0,C 180,E1 19494.332,E2 19494.332} C_VEL
LIN {X 0,Y 520.561,Z 247.883,A -85,B 0,C 180,E1 19490.891,E2 19490.891} C_VEL
LIN {X 0,Y 520.582,Z 247.89,A -85,B 0,C 180,E1 19487.465,E2 19487.465} C_VEL
LIN {X 0,Y 520.582,Z 247.885,A -85,B 0,C 180,E1 19483.928,E2 19483.928} C_VEL
LIN {X 0,Y 520.568,Z 247.88,A -85,B 0,C 180,E1 19480.479,E2 19480.479} C_VEL
LIN {X 0,Y 520.564,Z 247.882,A -85,B 0,C 180,E1 19476.953,E2 19476.953} C_VEL
LIN {X 0,Y 520.585,Z 247.889,A -85,B 0,C 180,E1 19473.449,E2 19473.449} C_VEL
LIN {X 0,Y 520.591,Z 247.876,A -85,B 0,C 180,E1 19469.956,E2 19469.956} C_VEL
LIN {X 0,Y 520.56,Z 247.883,A -85,B 0,C 180,E1 19466.487,E2 19466.487} C_VEL
LIN {X 0,Y 520.583,Z 247.891,A -85,B 0,C 180,E1 19463.066,E2 19463.066} C_VEL
LIN {X 0,Y 520.583,Z 247.878,A -85,B 0,C 180,E1 19459.639,E2 19459.639} C_VEL
LIN {X 0,Y 520.561,Z 247.886,A -85,B 0,C 180,E1 19456.17,E2 19456.17} C_VEL
LIN {X 0,Y 520.565,Z 247.89,A -85,B 0,C 180,E1 19452.647,E2 19452.647} C_VEL
LIN {X 0,Y 520.583,Z 247.884,A -85,B 0,C 180,E1 19449.172,E2 19449.172} C_VEL
LIN {X 0,Y 520.578,Z 247.885,A -85,B 0,C 180,E1 19445.731,E2 19445.731} C_VEL
LIN {X 0,Y 520.558,Z 247.885,A -85,B 0,C 180,E1 19442.311,E2 19442.311} C_VEL
LIN {X 0,Y 520.585,Z 247.887,A -85,B 0,C 180,E1 19438.899,E2 19438.899} C_VEL
LIN {X 0,Y 520.583,Z 247.884,A -85,B 0,C 180,E1 19435.372,E2 19435.372} C_VEL
LIN {X 0,Y 520.555,Z 247.883,A -85,B 0,C 180,E1 19431.939,E2 19431.939} C_VEL
LIN {X 0,Y 520.573,Z 247.883,A -85,B 0,C 180,E1 19428.477,E2 19428.477} C_VEL
LIN {X 0,Y 520.587,Z 247.888,A -85,B 0,C 180,E1 19424.972,E2 19424.972} C_VEL
LIN {X 0,Y 520.564,Z 247.887,A -85,B 0,C 180,E1 19421.523,E2 19421.523} C_VEL
LIN {X 0,Y 520.556,Z 247.891,A -85,B 0,C 180,E1 19418.003,E2 19418.003} C_VEL
LIN {X 0,Y 520.583,Z 247.883,A -85,B 0,C 180,E1 19414.639,E2 19414.639} C_VEL
LIN {X 0,Y 520.574,Z 247.88,A -85,B 0,C 180,E1 19411.177,E2 19411.177} C_VEL
LIN {X 0,Y 520.553,Z 247.888,A -85,B 0,C 180,E1 19407.725,E2 19407.725} C_VEL
LIN {X 0,Y 520.582,Z 247.887,A -85,B 0,C 180,E1 19404.276,E2 19404.276} C_VEL
LIN {X 0,Y 520.589,Z 247.888,A -85,B 0,C 180,E1 19400.81,E2 19400.81} C_VEL
LIN {X 0,Y 520.551,Z 247.888,A -85,B 0,C 180,E1 19397.459,E2 19397.459} C_VEL
LIN {X 0,Y 520.579,Z 247.89,A -85,B 0,C 180,E1 19394.047,E2 19394.047} C_VEL
LIN {X 0,Y 520.618,Z 248.112,A -85,B 0,C 180,E1 19392.567,E2 19392.567} C_VEL
LIN {X 0,Y 521.908,Z 251.377,A -85,B 0,C 180,E1 19392.149,E2 19392.149} C_VEL
LIN {X 0,Y 533.504,Z 276.694,A -85,B 0,C 180,E1 19389.322,E2 19389.322} C_VEL
LIN {X 0,Y 532.683,Z 302.627,A -85,B 0,C 180,E1 19387.64,E2 19387.64} C_VEL
LIN {X 0,Y 535.235,Z 319,A -85,B 0,C 180,E1 19387.173,E2 19387.173} C_VEL
LIN {X 0,Y 532.662,Z 536.527,A -85,B 0,C 180,E1 19383.849,E2 19383.849} C_VEL
LIN {X 0,Y 531.773,Z 609.44,A -85,B 0,C 180,E1 19382.721,E2 19382.721} C_VEL
LIN {X 0,Y 531.047,Z 631.086,A -85,B 0,C 180,E1 19382.187,E2 19382.187} C_VEL
LIN {X 0,Y 530.189,Z 653.251,A -85,B 0,C 180,E1 19381.427,E2 19381.427} C_VEL
LIN {X 0,Y 529.207,Z 673.415,A -85,B 0,C 180,E1 19380.545,E2 19380.545} C_VEL
LIN {X 0,Y 528.047,Z 693.865,A -85,B 0,C 180,E1 19379.423,E2 19379.423} C_VEL
LIN {X 0,Y 526.793,Z 714.149,A -85,B 0,C 180,E1 19378.079,E2 19378.079} C_VEL
LIN {X 0,Y 525.569,Z 733.453,A -85,B 0,C 180,E1 19376.554,E2 19376.554} C_VEL
LIN {X 0,Y 524.425,Z 751.13,A -85,B 0,C 180,E1 19374.919,E2 19374.919} C_VEL
LIN {X 0,Y 523.333,Z 767.71,A -85,B 0,C 180,E1 19373.116,E2 19373.116} C_VEL
LIN {X 0,Y 522.41,Z 782.882,A -85,B 0,C 180,E1 19371.205,E2 19371.205} C_VEL
LIN {X 0,Y 521.626,Z 797.058,A -85,B 0,C 180,E1 19369.132,E2 19369.132} C_VEL
LIN {X 0,Y 521.011,Z 809.736,A -85,B 0,C 180,E1 19366.958,E2 19366.958} C_VEL
LIN {X 0,Y 520.563,Z 820.337,A -85,B 0,C 180,E1 19364.799,E2 19364.799} C_VEL
LIN {X 0,Y 520.243,Z 830.076,A -85,B 0,C 180,E1 19362.429,E2 19362.429} C_VEL
LIN {X 0,Y 520.066,Z 837.71,A -85,B 0,C 180,E1 19360.149,E2 19360.149} C_VEL
LIN {X 0,Y 519.969,Z 843.656,A -85,B 0,C 180,E1 19357.846,E2 19357.846} C_VEL
LIN {X 0,Y 519.928,Z 848.305,A -85,B 0,C 180,E1 19355.406,E2 19355.406} C_VEL
LIN {X 0,Y 519.916,Z 851.012,A -85,B 0,C 180,E1 19353.196,E2 19353.196} C_VEL
LIN {X 0,Y 519.902,Z 852.351,A -85,B 0,C 180,E1 19350.77,E2 19350.77} C_VEL
LIN {X 0,Y 519.898,Z 852.149,A -85,B 0,C 180,E1 19348.456,E2 19348.456} C_VEL
LIN {X 0,Y 519.908,Z 850.331,A -85,B 0,C 180,E1 19346.139,E2 19346.139} C_VEL
LIN {X 0,Y 519.928,Z 846.807,A -85,B 0,C 180,E1 19343.706,E2 19343.706} C_VEL
LIN {X 0,Y 519.981,Z 841.869,A -85,B 0,C 180,E1 19341.373,E2 19341.373} C_VEL
LIN {X 0,Y 520.1,Z 835.464,A -85,B 0,C 180,E1 19339.14,E2 19339.14} C_VEL
LIN {X 0,Y 520.328,Z 827.052,A -85,B 0,C 180,E1 19336.78,E2 19336.78} C_VEL
LIN {X 0,Y 520.687,Z 817.216,A -85,B 0,C 180,E1 19334.518,E2 19334.518} C_VEL
LIN {X 0,Y 521.174,Z 805.911,A -85,B 0,C 180,E1 19332.354,E2 19332.354} C_VEL
LIN {X 0,Y 521.862,Z 792.542,A -85,B 0,C 180,E1 19330.174,E2 19330.174} C_VEL
LIN {X 0,Y 522.682,Z 778.57,A -85,B 0,C 180,E1 19328.215,E2 19328.215} C_VEL
LIN {X 0,Y 523.677,Z 762.528,A -85,B 0,C 180,E1 19326.29,E2 19326.29} C_VEL
LIN {X 0,Y 524.739,Z 745.927,A -85,B 0,C 180,E1 19324.579,E2 19324.579} C_VEL
LIN {X 0,Y 525.966,Z 727.116,A -85,B 0,C 180,E1 19322.916,E2 19322.916} C_VEL
LIN {X 0,Y 527.199,Z 708.419,A -85,B 0,C 180,E1 19321.511,E2 19321.511} C_VEL
LIN {X 0,Y 528.33,Z 688.721,A -85,B 0,C 180,E1 19320.274,E2 19320.274} C_VEL
LIN {X 0,Y 529.457,Z 668.299,A -85,B 0,C 180,E1 19319.217,E2 19319.217} C_VEL
LIN {X 0,Y 530.44,Z 647.672,A -85,B 0,C 180,E1 19318.353,E2 19318.353} C_VEL
LIN {X 0,Y 531.227,Z 626.714,A -85,B 0,C 180,E1 19317.691,E2 19317.691} C_VEL
LIN {X 0,Y 531.846,Z 604.202,A -85,B 0,C 180,E1 19317.186,E2 19317.186} C_VEL
LIN {X 0,Y 534.406,Z 386.218,A -85,B 0,C 180,E1 19313.863,E2 19313.863} C_VEL
LIN {X 0,Y 535.07,Z 316.763,A -85,B 0,C 180,E1 19312.776,E2 19312.776} C_VEL
LIN {X 0,Y 532.584,Z 301.282,A -85,B 0,C 180,E1 19312.3,E2 19312.3} C_VEL
LIN {X 0,Y 533.426,Z 276.586,A -85,B 0,C 180,E1 19310.687,E2 19310.687} C_VEL
LIN {X 0,Y 521.731,Z 251.118,A -85,B 0,C 180,E1 19307.873,E2 19307.873} C_VEL
LIN {X 0,Y 520.636,Z 248.225,A -85,B 0,C 180,E1 19307.515,E2 19307.515} C_VEL
LIN {X 0,Y 520.561,Z 247.887,A -85,B 0,C 180,E1 19306.859,E2 19306.859} C_VEL
LIN {X 0,Y 520.583,Z 247.878,A -85,B 0,C 180,E1 19303.44,E2 19303.44} C_VEL
LIN {X 0,Y 520.585,Z 247.889,A -85,B 0,C 180,E1 19299.904,E2 19299.904} C_VEL
LIN {X 0,Y 520.569,Z 247.891,A -85,B 0,C 180,E1 19296.406,E2 19296.406} C_VEL
LIN {X 0,Y 520.58,Z 247.887,A -85,B 0,C 180,E1 19292.926,E2 19292.926} C_VEL
LIN {X 0,Y 520.575,Z 247.885,A -85,B 0,C 180,E1 19289.453,E2 19289.453} C_VEL
LIN {X 0,Y 520.583,Z 247.888,A -85,B 0,C 180,E1 19285.971,E2 19285.971} C_VEL
LIN {X 0,Y 520.576,Z 247.887,A -85,B 0,C 180,E1 19282.472,E2 19282.472} C_VEL
LIN {X 0,Y 520.575,Z 247.887,A -85,B 0,C 180,E1 19279.058,E2 19279.058} C_VEL
LIN {X 0,Y 520.568,Z 247.89,A -85,B 0,C 180,E1 19275.599,E2 19275.599} C_VEL
LIN {X 0,Y 520.584,Z 247.892,A -85,B 0,C 180,E1 19272.145,E2 19272.145} C_VEL
LIN {X 0,Y 520.584,Z 247.886,A -85,B 0,C 180,E1 19268.617,E2 19268.617} C_VEL
LIN {X 0,Y 520.555,Z 247.886,A -85,B 0,C 180,E1 19265.18,E2 19265.18} C_VEL
LIN {X 0,Y 520.572,Z 247.888,A -85,B 0,C 180,E1 19261.762,E2 19261.762} C_VEL
LIN {X 0,Y 520.588,Z 247.885,A -85,B 0,C 180,E1 19258.35,E2 19258.35} C_VEL
LIN {X 0,Y 520.548,Z 247.889,A -85,B 0,C 180,E1 19254.932,E2 19254.932} C_VEL
LIN {X 0,Y 520.544,Z 247.892,A -85,B 0,C 180,E1 19251.384,E2 19251.384} C_VEL
LIN {X 0,Y 520.587,Z 247.888,A -85,B 0,C 180,E1 19248.029,E2 19248.029} C_VEL
LIN {X 0,Y 520.54,Z 247.892,A -85,B 0,C 180,E1 19244.744,E2 19244.744} C_VEL
LIN {X 0,Y 520.533,Z 247.895,A -85,B 0,C 180,E1 19241.259,E2 19241.259} C_VEL
LIN {X 0,Y 520.583,Z 247.881,A -85,B 0,C 180,E1 19237.888,E2 19237.888} C_VEL
LIN {X 0,Y 520.536,Z 247.883,A -85,B 0,C 180,E1 19234.517,E2 19234.517} C_VEL
LIN {X 0,Y 520.597,Z 248.163,A -85,B 0,C 180,E1 19233.695,E2 19233.695} C_VEL
LIN {X 0,Y 527.843,Z 266.12,A -85,B 0,C 180,E1 19231.366,E2 19231.366} C_VEL
LIN {X 0,Y 530.193,Z 272.723,A -85,B 0,C 180,E1 19230.578,E2 19230.578} C_VEL
LIN {X 0,Y 528.937,Z 299.786,A -85,B 0,C 180,E1 19228.363,E2 19228.363} C_VEL
LIN {X 0,Y 531.68,Z 315.638,A -85,B 0,C 180,E1 19227.885,E2 19227.885} C_VEL
LIN {X 0,Y 531.049,Z 362.988,A -85,B 0,C 180,E1 19227.164,E2 19227.164} C_VEL
LIN {X 0,Y 530.138,Z 370.681,A -85,B 0,C 180,E1 19227.107,E2 19227.107} C_VEL
LIN {X 0,Y 524.709,Z 391.215,A -85,B 0,C 180,E1 19227.174,E2 19227.174} C_VEL
LIN {X 0,Y 523.985,Z 397.819,A -85,B 0,C 180,E1 19227.121,E2 19227.121} C_VEL
LIN {X 0,Y 521.88,Z 561.791,A -85,B 0,C 180,E1 19224.606,E2 19224.606} C_VEL
LIN {X 0,Y 521.225,Z 582.597,A -85,B 0,C 180,E1 19224.079,E2 19224.079} C_VEL
LIN {X 0,Y 520.429,Z 601.895,A -85,B 0,C 180,E1 19223.386,E2 19223.386} C_VEL
LIN {X 0,Y 519.429,Z 621.451,A -85,B 0,C 180,E1 19222.474,E2 19222.474} C_VEL
LIN {X 0,Y 518.348,Z 640.393,A -85,B 0,C 180,E1 19221.373,E2 19221.373} C_VEL
LIN {X 0,Y 517.319,Z 658.361,A -85,B 0,C 180,E1 19220.114,E2 19220.114} C_VEL
LIN {X 0,Y 516.256,Z 675.6,A -85,B 0,C 180,E1 19218.669,E2 19218.669} C_VEL
LIN {X 0,Y 515.193,Z 692.581,A -85,B 0,C 180,E1 19216.968,E2 19216.968} C_VEL
LIN {X 0,Y 514.296,Z 707.411,A -85,B 0,C 180,E1 19215.204,E2 19215.204} C_VEL
LIN {X 0,Y 513.544,Z 720.776,A -85,B 0,C 180,E1 19213.332,E2 19213.332} C_VEL
LIN {X 0,Y 512.947,Z 733.01,A -85,B 0,C 180,E1 19211.303,E2 19211.303} C_VEL
LIN {X 0,Y 512.493,Z 743.898,A -85,B 0,C 180,E1 19209.135,E2 19209.135} C_VEL
LIN {X 0,Y 512.207,Z 752.842,A -85,B 0,C 180,E1 19206.959,E2 19206.959} C_VEL
LIN {X 0,Y 512.035,Z 760.059,A -85,B 0,C 180,E1 19204.765,E2 19204.765} C_VEL
LIN {X 0,Y 511.947,Z 765.74,A -85,B 0,C 180,E1 19202.468,E2 19202.468} C_VEL
LIN {X 0,Y 511.917,Z 769.519,A -85,B 0,C 180,E1 19200.26,E2 19200.26} C_VEL
LIN {X 0,Y 511.914,Z 771.814,A -85,B 0,C 180,E1 19197.955,E2 19197.955} C_VEL
LIN {X 0,Y 511.909,Z 772.455,A -85,B 0,C 180,E1 19195.698,E2 19195.698} C_VEL
LIN {X 0,Y 511.911,Z 771.527,A -85,B 0,C 180,E1 19193.482,E2 19193.482} C_VEL
LIN {X 0,Y 511.926,Z 769.025,A -85,B 0,C 180,E1 19191.303,E2 19191.303} C_VEL
LIN {X 0,Y 511.957,Z 764.826,A -85,B 0,C 180,E1 19189.036,E2 19189.036} C_VEL
LIN {X 0,Y 512.05,Z 759.007,A -85,B 0,C 180,E1 19186.799,E2 19186.799} C_VEL
LIN {X 0,Y 512.245,Z 751.514,A -85,B 0,C 180,E1 19184.585,E2 19184.585} C_VEL
LIN {X 0,Y 512.565,Z 742.166,A -85,B 0,C 180,E1 19182.392,E2 19182.392} C_VEL
LIN {X 0,Y 513.02,Z 731.481,A -85,B 0,C 180,E1 19180.33,E2 19180.33} C_VEL
LIN {X 0,Y 513.612,Z 719.562,A -85,B 0,C 180,E1 19178.397,E2 19178.397} C_VEL
LIN {X 0,Y 514.404,Z 705.561,A -85,B 0,C 180,E1 19176.474,E2 19176.474} C_VEL
LIN {X 0,Y 515.305,Z 690.591,A -85,B 0,C 180,E1 19174.731,E2 19174.731} C_VEL
LIN {X 0,Y 516.334,Z 674.131,A -85,B 0,C 180,E1 19173.109,E2 19173.109} C_VEL
LIN {X 0,Y 517.431,Z 656.65,A -85,B 0,C 180,E1 19171.662,E2 19171.662} C_VEL
LIN {X 0,Y 518.505,Z 638.069,A -85,B 0,C 180,E1 19170.388,E2 19170.388} C_VEL
LIN {X 0,Y 519.581,Z 618.502,A -85,B 0,C 180,E1 19169.284,E2 19169.284} C_VEL
LIN {X 0,Y 520.505,Z 599.497,A -85,B 0,C 180,E1 19168.433,E2 19168.433} C_VEL
LIN {X 0,Y 521.313,Z 578.686,A -85,B 0,C 180,E1 19167.726,E2 19167.726} C_VEL
LIN {X 0,Y 521.894,Z 557.94,A -85,B 0,C 180,E1 19167.242,E2 19167.242} C_VEL
LIN {X 0,Y 524.92,Z 315.981,A -85,B 0,C 180,E1 19163.559,E2 19163.559} C_VEL
LIN {X 0,Y 521.844,Z 299.017,A -85,B 0,C 180,E1 19163.013,E2 19163.013} C_VEL
LIN {X 0,Y 522.947,Z 275.298,A -85,B 0,C 180,E1 19161.037,E2 19161.037} C_VEL
LIN {X 0,Y 516.462,Z 258.62,A -85,B 0,C 180,E1 19158.964,E2 19158.964} C_VEL
LIN {X 0,Y 512.676,Z 249.159,A -85,B 0,C 180,E1 19157.703,E2 19157.703} C_VEL
LIN {X 0,Y 512.645,Z 248.85,A -85,B 0,C 180,E1 19155.891,E2 19155.891} C_VEL
LIN {X 0,Y 512.639,Z 248.855,A -85,B 0,C 180,E1 19152.405,E2 19152.405} C_VEL
LIN {X 0,Y 512.633,Z 248.878,A -85,B 0,C 180,E1 19148.97,E2 19148.97} C_VEL
LIN {X 0,Y 512.628,Z 248.857,A -85,B 0,C 180,E1 19145.454,E2 19145.454} C_VEL
LIN {X 0,Y 512.643,Z 248.875,A -85,B 0,C 180,E1 19141.964,E2 19141.964} C_VEL
LIN {X 0,Y 512.646,Z 248.871,A -85,B 0,C 180,E1 19138.462,E2 19138.462} C_VEL
LIN {X 0,Y 512.624,Z 248.872,A -85,B 0,C 180,E1 19135.002,E2 19135.002} C_VEL
LIN {X 0,Y 512.643,Z 248.876,A -85,B 0,C 180,E1 19131.452,E2 19131.452} C_VEL
LIN {X 0,Y 512.641,Z 248.877,A -85,B 0,C 180,E1 19127.994,E2 19127.994} C_VEL
LIN {X 0,Y 512.629,Z 248.874,A -85,B 0,C 180,E1 19124.599,E2 19124.599} C_VEL
LIN {X 0,Y 512.631,Z 248.87,A -85,B 0,C 180,E1 19121.092,E2 19121.092} C_VEL
LIN {X 0,Y 512.644,Z 248.878,A -85,B 0,C 180,E1 19117.622,E2 19117.622} C_VEL
LIN {X 0,Y 512.641,Z 248.872,A -85,B 0,C 180,E1 19114.173,E2 19114.173} C_VEL
LIN {X 0,Y 512.622,Z 248.869,A -85,B 0,C 180,E1 19110.669,E2 19110.669} C_VEL
LIN {X 0,Y 512.643,Z 248.878,A -85,B 0,C 180,E1 19107.153,E2 19107.153} C_VEL
LIN {X 0,Y 512.645,Z 248.87,A -85,B 0,C 180,E1 19103.688,E2 19103.688} C_VEL
LIN {X 0,Y 512.623,Z 248.867,A -85,B 0,C 180,E1 19100.257,E2 19100.257} C_VEL
LIN {X 0,Y 512.628,Z 248.879,A -85,B 0,C 180,E1 19096.736,E2 19096.736} C_VEL
LIN {X 0,Y 512.643,Z 248.865,A -85,B 0,C 180,E1 19093.291,E2 19093.291} C_VEL
LIN {X 0,Y 512.639,Z 248.872,A -85,B 0,C 180,E1 19089.768,E2 19089.768} C_VEL
LIN {X 0,Y 512.618,Z 248.878,A -85,B 0,C 180,E1 19086.27,E2 19086.27} C_VEL
LIN {X 0,Y 512.639,Z 248.869,A -85,B 0,C 180,E1 19082.794,E2 19082.794} C_VEL
LIN {X 0,Y 512.65,Z 248.875,A -85,B 0,C 180,E1 19079.329,E2 19079.329} C_VEL
LIN {X 0,Y 512.621,Z 248.875,A -85,B 0,C 180,E1 19075.861,E2 19075.861} C_VEL
LIN {X 0,Y 512.62,Z 248.872,A -85,B 0,C 180,E1 19072.265,E2 19072.265} C_VEL
LIN {X 0,Y 512.647,Z 248.876,A -85,B 0,C 180,E1 19068.816,E2 19068.816} C_VEL
LIN {X 0,Y 512.644,Z 248.875,A -85,B 0,C 180,E1 19065.312,E2 19065.312} C_VEL
LIN {X 0,Y 512.617,Z 248.878,A -85,B 0,C 180,E1 19061.815,E2 19061.815} C_VEL
LIN {X 0,Y 512.639,Z 248.873,A -85,B 0,C 180,E1 19058.368,E2 19058.368} C_VEL
LIN {X 0,Y 512.646,Z 248.871,A -85,B 0,C 180,E1 19054.837,E2 19054.837} C_VEL
LIN {X 0,Y 512.623,Z 248.87,A -85,B 0,C 180,E1 19051.364,E2 19051.364} C_VEL
LIN {X 0,Y 512.616,Z 248.876,A -85,B 0,C 180,E1 19047.826,E2 19047.826} C_VEL
LIN {X 0,Y 512.645,Z 248.874,A -85,B 0,C 180,E1 19044.326,E2 19044.326} C_VEL
LIN {X 0,Y 512.65,Z 248.877,A -85,B 0,C 180,E1 19040.808,E2 19040.808} C_VEL
LIN {X 0,Y 512.612,Z 248.876,A -85,B 0,C 180,E1 19037.403,E2 19037.403} C_VEL
LIN {X 0,Y 512.635,Z 248.88,A -85,B 0,C 180,E1 19033.969,E2 19033.969} C_VEL
LIN {X 0,Y 512.654,Z 249.159,A -85,B 0,C 180,E1 19033.246,E2 19033.246} C_VEL
LIN {X 0,Y 513.949,Z 252.354,A -85,B 0,C 180,E1 19032.825,E2 19032.825} C_VEL
LIN {X 0,Y 524.868,Z 276.072,A -85,B 0,C 180,E1 19030.08,E2 19030.08} C_VEL
LIN {X 0,Y 526.698,Z 280.265,A -85,B 0,C 180,E1 19029.629,E2 19029.629} C_VEL
LIN {X 0,Y 525.913,Z 302.719,A -85,B 0,C 180,E1 19028.16,E2 19028.16} C_VEL
LIN {X 0,Y 528.694,Z 320.442,A -85,B 0,C 180,E1 19027.653,E2 19027.653} C_VEL
LIN {X 0,Y 526.151,Z 526.721,A -85,B 0,C 180,E1 19024.485,E2 19024.485} C_VEL
LIN {X 0,Y 525.046,Z 609.243,A -85,B 0,C 180,E1 19023.198,E2 19023.198} C_VEL
LIN {X 0,Y 524.276,Z 630.68,A -85,B 0,C 180,E1 19022.667,E2 19022.667} C_VEL
LIN {X 0,Y 523.346,Z 652.507,A -85,B 0,C 180,E1 19021.918,E2 19021.918} C_VEL
LIN {X 0,Y 522.31,Z 672.189,A -85,B 0,C 180,E1 19021.056,E2 19021.056} C_VEL
LIN {X 0,Y 521.075,Z 691.772,A -85,B 0,C 180,E1 19019.989,E2 19019.989} C_VEL
LIN {X 0,Y 519.708,Z 712.523,A -85,B 0,C 180,E1 19018.621,E2 19018.621} C_VEL
LIN {X 0,Y 518.439,Z 730.772,A -85,B 0,C 180,E1 19017.197,E2 19017.197} C_VEL
LIN {X 0,Y 517.11,Z 748.718,A -85,B 0,C 180,E1 19015.541,E2 19015.541} C_VEL
LIN {X 0,Y 515.899,Z 765.683,A -85,B 0,C 180,E1 19013.711,E2 19013.711} C_VEL
LIN {X 0,Y 514.846,Z 781.185,A -85,B 0,C 180,E1 19011.772,E2 19011.772} C_VEL
LIN {X 0,Y 513.942,Z 795.639,A -85,B 0,C 180,E1 19009.666,E2 19009.666} C_VEL
LIN {X 0,Y 513.204,Z 808.465,A -85,B 0,C 180,E1 19007.458,E2 19007.458} C_VEL
LIN {X 0,Y 512.664,Z 819.821,A -85,B 0,C 180,E1 19005.148,E2 19005.148} C_VEL
LIN {X 0,Y 512.315,Z 829.262,A -85,B 0,C 180,E1 19002.854,E2 19002.854} C_VEL
LIN {X 0,Y 512.102,Z 836.886,A -85,B 0,C 180,E1 19000.574,E2 19000.574} C_VEL
LIN {X 0,Y 511.988,Z 843.148,A -85,B 0,C 180,E1 18998.195,E2 18998.195} C_VEL
LIN {X 0,Y 511.928,Z 847.825,A -85,B 0,C 180,E1 18995.828,E2 18995.828} C_VEL
LIN {X 0,Y 511.911,Z 850.788,A -85,B 0,C 180,E1 18993.47,E2 18993.47} C_VEL
LIN {X 0,Y 511.912,Z 852.305,A -85,B 0,C 180,E1 18991.006,E2 18991.006} C_VEL
LIN {X 0,Y 511.905,Z 852.236,A -85,B 0,C 180,E1 18988.656,E2 18988.656} C_VEL
LIN {X 0,Y 511.907,Z 850.558,A -85,B 0,C 180,E1 18986.303,E2 18986.303} C_VEL
LIN {X 0,Y 511.933,Z 847.424,A -85,B 0,C 180,E1 18983.945,E2 18983.945} C_VEL
LIN {X 0,Y 511.989,Z 842.888,A -85,B 0,C 180,E1 18981.69,E2 18981.69} C_VEL
LIN {X 0,Y 512.111,Z 836.172,A -85,B 0,C 180,E1 18979.196,E2 18979.196} C_VEL
LIN {X 0,Y 512.35,Z 828.194,A -85,B 0,C 180,E1 18976.857,E2 18976.857} C_VEL
LIN {X 0,Y 512.71,Z 818.775,A -85,B 0,C 180,E1 18974.619,E2 18974.619} C_VEL
LIN {X 0,Y 513.276,Z 807.045,A -85,B 0,C 180,E1 18972.282,E2 18972.282} C_VEL
LIN {X 0,Y 514.021,Z 794.09,A -85,B 0,C 180,E1 18970.097,E2 18970.097} C_VEL
LIN {X 0,Y 514.965,Z 779.467,A -85,B 0,C 180,E1 18967.991,E2 18967.991} C_VEL
LIN {X 0,Y 516.047,Z 763.635,A -85,B 0,C 180,E1 18966.051,E2 18966.051} C_VEL
LIN {X 0,Y 517.262,Z 746.663,A -85,B 0,C 180,E1 18964.26,E2 18964.26} C_VEL
LIN {X 0,Y 518.571,Z 728.574,A -85,B 0,C 180,E1 18962.621,E2 18962.621} C_VEL
LIN {X 0,Y 519.9,Z 710.06,A -85,B 0,C 180,E1 18961.199,E2 18961.199} C_VEL
LIN {X 0,Y 521.142,Z 690.728,A -85,B 0,C 180,E1 18959.949,E2 18959.949} C_VEL
LIN {X 0,Y 522.417,Z 670.097,A -85,B 0,C 180,E1 18958.846,E2 18958.846} C_VEL
LIN {X 0,Y 523.435,Z 650.694,A -85,B 0,C 180,E1 18958.008,E2 18958.008} C_VEL
LIN {X 0,Y 524.338,Z 629.319,A -85,B 0,C 180,E1 18957.295,E2 18957.295} C_VEL
LIN {X 0,Y 525.069,Z 607.827,A -85,B 0,C 180,E1 18956.777,E2 18956.777} C_VEL
LIN {X 0,Y 527.84,Z 393.655,A -85,B 0,C 180,E1 18953.466,E2 18953.466} C_VEL
LIN {X 0,Y 528.49,Z 318.191,A -85,B 0,C 180,E1 18952.303,E2 18952.303} C_VEL
LIN {X 0,Y 525.753,Z 301.891,A -85,B 0,C 180,E1 18951.823,E2 18951.823} C_VEL
LIN {X 0,Y 526.44,Z 279.713,A -85,B 0,C 180,E1 18950.344,E2 18950.344} C_VEL
LIN {X 0,Y 514.227,Z 252.751,A -85,B 0,C 180,E1 18947.306,E2 18947.306} C_VEL
LIN {X 0,Y 512.668,Z 249.191,A -85,B 0,C 180,E1 18946.838,E2 18946.838} C_VEL
LIN {X 0,Y 512.645,Z 248.864,A -85,B 0,C 180,E1 18945.869,E2 18945.869} C_VEL
LIN {X 0,Y 512.622,Z 248.866,A -85,B 0,C 180,E1 18942.444,E2 18942.444} C_VEL
LIN {X 0,Y 512.636,Z 248.878,A -85,B 0,C 180,E1 18938.906,E2 18938.906} C_VEL
LIN {X 0,Y 512.641,Z 248.879,A -85,B 0,C 180,E1 18935.4,E2 18935.4} C_VEL
LIN {X 0,Y 512.645,Z 248.877,A -85,B 0,C 180,E1 18931.908,E2 18931.908} C_VEL
LIN {X 0,Y 512.634,Z 248.875,A -85,B 0,C 180,E1 18928.399,E2 18928.399} C_VEL
LIN {X 0,Y 512.646,Z 248.875,A -85,B 0,C 180,E1 18924.914,E2 18924.914} C_VEL
LIN {X 0,Y 512.631,Z 248.875,A -85,B 0,C 180,E1 18921.392,E2 18921.392} C_VEL
LIN {X 0,Y 512.64,Z 248.875,A -85,B 0,C 180,E1 18917.832,E2 18917.832} C_VEL
LIN {X 0,Y 512.642,Z 248.875,A -85,B 0,C 180,E1 18914.342,E2 18914.342} C_VEL
LIN {X 0,Y 512.633,Z 248.87,A -85,B 0,C 180,E1 18910.906,E2 18910.906} C_VEL
LIN {X 0,Y 512.618,Z 248.879,A -85,B 0,C 180,E1 18907.397,E2 18907.397} C_VEL
LIN {X 0,Y 512.641,Z 248.877,A -85,B 0,C 180,E1 18903.915,E2 18903.915} C_VEL
LIN {X 0,Y 512.65,Z 248.874,A -85,B 0,C 180,E1 18900.448,E2 18900.448} C_VEL
LIN {X 0,Y 512.61,Z 248.88,A -85,B 0,C 180,E1 18896.982,E2 18896.982} C_VEL
LIN {X 0,Y 512.606,Z 248.878,A -85,B 0,C 180,E1 18893.393,E2 18893.393} C_VEL
LIN {X 0,Y 512.646,Z 248.876,A -85,B 0,C 180,E1 18890.005,E2 18890.005} C_VEL
LIN {X 0,Y 512.616,Z 248.881,A -85,B 0,C 180,E1 18886.58,E2 18886.58} C_VEL
LIN {X 0,Y 512.593,Z 248.883,A -85,B 0,C 180,E1 18883.222,E2 18883.222} C_VEL
LIN {X 0,Y 512.642,Z 248.878,A -85,B 0,C 180,E1 18879.925,E2 18879.925} C_VEL
LIN {X 0,Y 512.591,Z 248.872,A -85,B 0,C 180,E1 18876.675,E2 18876.675} C_VEL
LIN {X 0,Y 512.647,Z 249.139,A -85,B 0,C 180,E1 18874.373,E2 18874.373} C_VEL
LIN {X 0,Y 520.509,Z 268.441,A -85,B 0,C 180,E1 18871.802,E2 18871.802} C_VEL
LIN {X 0,Y 523.291,Z 276.372,A -85,B 0,C 180,E1 18870.843,E2 18870.843} C_VEL
LIN {X 0,Y 522.102,Z 299.87,A -85,B 0,C 180,E1 18868.898,E2 18868.898} C_VEL
LIN {X 0,Y 525.121,Z 316.952,A -85,B 0,C 180,E1 18868.368,E2 18868.368} C_VEL
LIN {X 0,Y 523.985,Z 397.819,A -85,B 0,C 180,E1 18867.121,E2 18867.121} C_VEL
LIN {X 0,Y 523.035,Z 405.514,A -85,B 0,C 180,E1 18867.066,E2 18867.066} C_VEL
LIN {X 0,Y 517.567,Z 426.038,A -85,B 0,C 180,E1 18867.137,E2 18867.137} C_VEL
LIN {X 0,Y 516.875,Z 432.639,A -85,B 0,C 180,E1 18867.081,E2 18867.081} C_VEL
LIN {X 0,Y 515.006,Z 562.605,A -85,B 0,C 180,E1 18865.05,E2 18865.05} C_VEL
LIN {X 0,Y 514.3,Z 583.516,A -85,B 0,C 180,E1 18864.51,E2 18864.51} C_VEL
LIN {X 0,Y 513.483,Z 601.844,A -85,B 0,C 180,E1 18863.845,E2 18863.845} C_VEL
LIN {X 0,Y 512.394,Z 621.589,A -85,B 0,C 180,E1 18862.919,E2 18862.919} C_VEL
LIN {X 0,Y 511.229,Z 640.097,A -85,B 0,C 180,E1 18861.829,E2 18861.829} C_VEL
LIN {X 0,Y 510.026,Z 657.665,A -85,B 0,C 180,E1 18860.569,E2 18860.569} C_VEL
LIN {X 0,Y 508.685,Z 676.184,A -85,B 0,C 180,E1 18858.968,E2 18858.968} C_VEL
LIN {X 0,Y 507.558,Z 692.668,A -85,B 0,C 180,E1 18857.29,E2 18857.29} C_VEL
LIN {X 0,Y 506.546,Z 707.912,A -85,B 0,C 180,E1 18855.445,E2 18855.445} C_VEL
LIN {X 0,Y 505.719,Z 721.188,A -85,B 0,C 180,E1 18853.546,E2 18853.546} C_VEL
LIN {X 0,Y 505.059,Z 733.343,A -85,B 0,C 180,E1 18851.487,E2 18851.487} C_VEL
LIN {X 0,Y 504.557,Z 744.176,A -85,B 0,C 180,E1 18849.283,E2 18849.283} C_VEL
LIN {X 0,Y 504.238,Z 753.064,A -85,B 0,C 180,E1 18847.072,E2 18847.072} C_VEL
LIN {X 0,Y 504.047,Z 760.227,A -85,B 0,C 180,E1 18844.842,E2 18844.842} C_VEL
LIN {X 0,Y 503.953,Z 765.851,A -85,B 0,C 180,E1 18842.522,E2 18842.522} C_VEL
LIN {X 0,Y 503.918,Z 769.609,A -85,B 0,C 180,E1 18840.265,E2 18840.265} C_VEL
LIN {X 0,Y 503.914,Z 771.852,A -85,B 0,C 180,E1 18837.923,E2 18837.923} C_VEL
LIN {X 0,Y 503.908,Z 772.443,A -85,B 0,C 180,E1 18835.631,E2 18835.631} C_VEL
LIN {X 0,Y 503.914,Z 771.487,A -85,B 0,C 180,E1 18833.382,E2 18833.382} C_VEL
LIN {X 0,Y 503.928,Z 768.771,A -85,B 0,C 180,E1 18831.048,E2 18831.048} C_VEL
LIN {X 0,Y 503.963,Z 764.433,A -85,B 0,C 180,E1 18828.749,E2 18828.749} C_VEL
LIN {X 0,Y 504.091,Z 758.108,A -85,B 0,C 180,E1 18826.36,E2 18826.36} C_VEL
LIN {X 0,Y 504.324,Z 750.372,A -85,B 0,C 180,E1 18824.115,E2 18824.115} C_VEL
LIN {X 0,Y 504.677,Z 741.405,A -85,B 0,C 180,E1 18822.008,E2 18822.008} C_VEL
LIN {X 0,Y 505.25,Z 729.812,A -85,B 0,C 180,E1 18819.776,E2 18819.776} C_VEL
LIN {X 0,Y 505.979,Z 716.972,A -85,B 0,C 180,E1 18817.724,E2 18817.724} C_VEL
LIN {X 0,Y 506.835,Z 703.382,A -85,B 0,C 180,E1 18815.889,E2 18815.889} C_VEL
LIN {X 0,Y 507.867,Z 687.992,A -85,B 0,C 180,E1 18814.122,E2 18814.122} C_VEL
LIN {X 0,Y 509.082,Z 670.421,A -85,B 0,C 180,E1 18812.421,E2 18812.421} C_VEL
LIN {X 0,Y 510.354,Z 652.485,A -85,B 0,C 180,E1 18810.955,E2 18810.955} C_VEL
LIN {X 0,Y 511.576,Z 634.247,A -85,B 0,C 180,E1 18809.721,E2 18809.721} C_VEL
LIN {X 0,Y 512.693,Z 616.07,A -85,B 0,C 180,E1 18808.716,E2 18808.716} C_VEL
LIN {X 0,Y 513.672,Z 596.294,A -85,B 0,C 180,E1 18807.854,E2 18807.854} C_VEL
LIN {X 0,Y 514.486,Z 576.467,A -85,B 0,C 180,E1 18807.212,E2 18807.212} C_VEL
LIN {X 0,Y 515.043,Z 555.763,A -85,B 0,C 180,E1 18806.749,E2 18806.749} C_VEL
LIN {X 0,Y 518.327,Z 317.396,A -85,B 0,C 180,E1 18803.077,E2 18803.077} C_VEL
LIN {X 0,Y 514.984,Z 298.995,A -85,B 0,C 180,E1 18802.471,E2 18802.471} C_VEL
LIN {X 0,Y 516.039,Z 278.593,A -85,B 0,C 180,E1 18800.747,E2 18800.747} C_VEL
LIN {X 0,Y 508.949,Z 260.375,A -85,B 0,C 180,E1 18798.442,E2 18798.442} C_VEL
LIN {X 0,Y 504.741,Z 250.173,A -85,B 0,C 180,E1 18797.04,E2 18797.04} C_VEL
LIN {X 0,Y 504.702,Z 249.836,A -85,B 0,C 180,E1 18796.096,E2 18796.096} C_VEL
LIN {X 0,Y 504.703,Z 249.844,A -85,B 0,C 180,E1 18792.595,E2 18792.595} C_VEL
LIN {X 0,Y 504.69,Z 249.868,A -85,B 0,C 180,E1 18789.11,E2 18789.11} C_VEL
LIN {X 0,Y 504.693,Z 249.842,A -85,B 0,C 180,E1 18785.542,E2 18785.542} C_VEL
LIN {X 0,Y 504.703,Z 249.864,A -85,B 0,C 180,E1 18782.071,E2 18782.071} C_VEL
LIN {X 0,Y 504.703,Z 249.861,A -85,B 0,C 180,E1 18778.601,E2 18778.601} C_VEL
LIN {X 0,Y 504.686,Z 249.861,A -85,B 0,C 180,E1 18775.074,E2 18775.074} C_VEL
LIN {X 0,Y 504.707,Z 249.864,A -85,B 0,C 180,E1 18771.489,E2 18771.489} C_VEL
LIN {X 0,Y 504.703,Z 249.866,A -85,B 0,C 180,E1 18767.966,E2 18767.966} C_VEL
LIN {X 0,Y 504.694,Z 249.862,A -85,B 0,C 180,E1 18764.506,E2 18764.506} C_VEL
LIN {X 0,Y 504.687,Z 249.858,A -85,B 0,C 180,E1 18760.975,E2 18760.975} C_VEL
LIN {X 0,Y 504.705,Z 249.868,A -85,B 0,C 180,E1 18757.59,E2 18757.59} C_VEL
LIN {X 0,Y 504.703,Z 249.861,A -85,B 0,C 180,E1 18754.099,E2 18754.099} C_VEL
LIN {X 0,Y 504.684,Z 249.857,A -85,B 0,C 180,E1 18750.606,E2 18750.606} C_VEL
LIN {X 0,Y 504.702,Z 249.866,A -85,B 0,C 180,E1 18747.105,E2 18747.105} C_VEL
LIN {X 0,Y 504.706,Z 249.86,A -85,B 0,C 180,E1 18743.588,E2 18743.588} C_VEL
LIN {X 0,Y 504.691,Z 249.855,A -85,B 0,C 180,E1 18740.112,E2 18740.112} C_VEL
LIN {X 0,Y 504.683,Z 249.867,A -85,B 0,C 180,E1 18736.575,E2 18736.575} C_VEL
LIN {X 0,Y 504.706,Z 249.854,A -85,B 0,C 180,E1 18733.168,E2 18733.168} C_VEL
LIN {X 0,Y 504.706,Z 249.861,A -85,B 0,C 180,E1 18729.578,E2 18729.578} C_VEL
LIN {X 0,Y 504.681,Z 249.866,A -85,B 0,C 180,E1 18726.14,E2 18726.14} C_VEL
LIN {X 0,Y 504.692,Z 249.859,A -85,B 0,C 180,E1 18722.611,E2 18722.611} C_VEL
LIN {X 0,Y 504.707,Z 249.867,A -85,B 0,C 180,E1 18719.091,E2 18719.091} C_VEL
LIN {X 0,Y 504.696,Z 249.862,A -85,B 0,C 180,E1 18715.568,E2 18715.568} C_VEL
LIN {X 0,Y 504.679,Z 249.86,A -85,B 0,C 180,E1 18712.119,E2 18712.119} C_VEL
LIN {X 0,Y 504.705,Z 249.862,A -85,B 0,C 180,E1 18708.689,E2 18708.689} C_VEL
LIN {X 0,Y 504.712,Z 249.864,A -85,B 0,C 180,E1 18705.177,E2 18705.177} C_VEL
LIN {X 0,Y 504.681,Z 249.866,A -85,B 0,C 180,E1 18701.638,E2 18701.638} C_VEL
LIN {X 0,Y 504.684,Z 249.866,A -85,B 0,C 180,E1 18698.132,E2 18698.132} C_VEL
LIN {X 0,Y 504.706,Z 249.859,A -85,B 0,C 180,E1 18694.664,E2 18694.664} C_VEL
LIN {X 0,Y 504.701,Z 249.857,A -85,B 0,C 180,E1 18691.117,E2 18691.117} C_VEL
LIN {X 0,Y 504.675,Z 249.865,A -85,B 0,C 180,E1 18687.661,E2 18687.661} C_VEL
LIN {X 0,Y 504.695,Z 249.866,A -85,B 0,C 180,E1 18684.12,E2 18684.12} C_VEL
LIN {X 0,Y 504.711,Z 249.868,A -85,B 0,C 180,E1 18680.586,E2 18680.586} C_VEL
LIN {X 0,Y 504.682,Z 249.854,A -85,B 0,C 180,E1 18677.139,E2 18677.139} C_VEL
LIN {X 0,Y 504.729,Z 250.107,A -85,B 0,C 180,E1 18673.972,E2 18673.972} C_VEL
LIN {X 0,Y 506.031,Z 253.423,A -85,B 0,C 180,E1 18673.518,E2 18673.518} C_VEL
LIN {X 0,Y 513.592,Z 269.665,A -85,B 0,C 180,E1 18671.535,E2 18671.535} C_VEL
LIN {X 0,Y 519.92,Z 283.576,A -85,B 0,C 180,E1 18669.963,E2 18669.963} C_VEL
LIN {X 0,Y 519.174,Z 302.678,A -85,B 0,C 180,E1 18668.697,E2 18668.697} C_VEL
LIN {X 0,Y 522.143,Z 321.918,A -85,B 0,C 180,E1 18668.138,E2 18668.138} C_VEL
LIN {X 0,Y 519.4,Z 537.927,A -85,B 0,C 180,E1 18664.813,E2 18664.813} C_VEL
LIN {X 0,Y 518.34,Z 609.626,A -85,B 0,C 180,E1 18663.676,E2 18663.676} C_VEL
LIN {X 0,Y 517.513,Z 630.952,A -85,B 0,C 180,E1 18663.14,E2 18663.14} C_VEL
LIN {X 0,Y 516.501,Z 652.504,A -85,B 0,C 180,E1 18662.392,E2 18662.392} C_VEL
LIN {X 0,Y 515.382,Z 672.192,A -85,B 0,C 180,E1 18661.521,E2 18661.521} C_VEL
LIN {X 0,Y 514.034,Z 691.769,A -85,B 0,C 180,E1 18660.443,E2 18660.443} C_VEL
LIN {X 0,Y 512.545,Z 712.519,A -85,B 0,C 180,E1 18659.059,E2 18659.059} C_VEL
LIN {X 0,Y 511.128,Z 730.907,A -85,B 0,C 180,E1 18657.606,E2 18657.606} C_VEL
LIN {X 0,Y 509.696,Z 748.718,A -85,B 0,C 180,E1 18655.94,E2 18655.94} C_VEL
LIN {X 0,Y 508.387,Z 765.235,A -85,B 0,C 180,E1 18654.138,E2 18654.138} C_VEL
LIN {X 0,Y 507.247,Z 780.336,A -85,B 0,C 180,E1 18652.237,E2 18652.237} C_VEL
LIN {X 0,Y 506.225,Z 794.875,A -85,B 0,C 180,E1 18650.099,E2 18650.099} C_VEL
LIN {X 0,Y 505.418,Z 807.548,A -85,B 0,C 180,E1 18647.908,E2 18647.908} C_VEL
LIN {X 0,Y 504.787,Z 819.305,A -85,B 0,C 180,E1 18645.508,E2 18645.508} C_VEL
LIN {X 0,Y 504.382,Z 828.855,A -85,B 0,C 180,E1 18643.176,E2 18643.176} C_VEL
LIN {X 0,Y 504.129,Z 836.533,A -85,B 0,C 180,E1 18640.859,E2 18640.859} C_VEL
LIN {X 0,Y 503.994,Z 843.148,A -85,B 0,C 180,E1 18638.326,E2 18638.326} C_VEL
LIN {X 0,Y 503.93,Z 847.825,A -85,B 0,C 180,E1 18635.921,E2 18635.921} C_VEL
LIN {X 0,Y 503.91,Z 850.788,A -85,B 0,C 180,E1 18633.525,E2 18633.525} C_VEL
LIN {X 0,Y 503.912,Z 852.305,A -85,B 0,C 180,E1 18631.022,E2 18631.022} C_VEL
LIN {X 0,Y 503.908,Z 852.259,A -85,B 0,C 180,E1 18628.748,E2 18628.748} C_VEL
LIN {X 0,Y 503.907,Z 850.671,A -85,B 0,C 180,E1 18626.358,E2 18626.358} C_VEL
LIN {X 0,Y 503.935,Z 847.63,A -85,B 0,C 180,E1 18623.963,E2 18623.963} C_VEL
LIN {X 0,Y 503.992,Z 842.888,A -85,B 0,C 180,E1 18621.557,E2 18621.557} C_VEL
LIN {X 0,Y 504.137,Z 836.171,A -85,B 0,C 180,E1 18619.023,E2 18619.023} C_VEL
LIN {X 0,Y 504.4,Z 828.424,A -85,B 0,C 180,E1 18616.705,E2 18616.705} C_VEL
LIN {X 0,Y 504.818,Z 818.775,A -85,B 0,C 180,E1 18614.372,E2 18614.372} C_VEL
LIN {X 0,Y 505.441,Z 807.181,A -85,B 0,C 180,E1 18612.024,E2 18612.024} C_VEL
LIN {X 0,Y 506.225,Z 794.859,A -85,B 0,C 180,E1 18609.898,E2 18609.898} C_VEL
LIN {X 0,Y 507.249,Z 780.318,A -85,B 0,C 180,E1 18607.761,E2 18607.761} C_VEL
LIN {X 0,Y 508.433,Z 764.648,A -85,B 0,C 180,E1 18605.793,E2 18605.793} C_VEL
LIN {X 0,Y 509.84,Z 746.927,A -85,B 0,C 180,E1 18603.884,E2 18603.884} C_VEL
LIN {X 0,Y 511.239,Z 729.303,A -85,B 0,C 180,E1 18602.258,E2 18602.258} C_VEL
LIN {X 0,Y 512.681,Z 710.868,A -85,B 0,C 180,E1 18600.818,E2 18600.818} C_VEL
LIN {X 0,Y 514.039,Z 691.73,A -85,B 0,C 180,E1 18599.555,E2 18599.555} C_VEL
LIN {X 0,Y 515.386,Z 672.139,A -85,B 0,C 180,E1 18598.476,E2 18598.476} C_VEL
LIN {X 0,Y 516.543,Z 651.715,A -85,B 0,C 180,E1 18597.575,E2 18597.575} C_VEL
LIN {X 0,Y 517.565,Z 629.891,A -85,B 0,C 180,E1 18596.83,E2 18596.83} C_VEL
LIN {X 0,Y 518.363,Z 608.576,A -85,B 0,C 180,E1 18596.305,E2 18596.305} C_VEL
LIN {X 0,Y 520.03,Z 489.867,A -85,B 0,C 180,E1 18594.449,E2 18594.449} C_VEL
LIN {X 0,Y 521.958,Z 319.992,A -85,B 0,C 180,E1 18591.837,E2 18591.837} C_VEL
LIN {X 0,Y 518.97,Z 301.708,A -85,B 0,C 180,E1 18591.287,E2 18591.287} C_VEL
LIN {X 0,Y 519.736,Z 283.369,A -85,B 0,C 180,E1 18590.052,E2 18590.052} C_VEL
LIN {X 0,Y 507.949,Z 257.432,A -85,B 0,C 180,E1 18587.071,E2 18587.071} C_VEL
LIN {X 0,Y 504.772,Z 250.348,A -85,B 0,C 180,E1 18586.177,E2 18586.177} C_VEL
LIN {X 0,Y 504.706,Z 249.865,A -85,B 0,C 180,E1 18585.943,E2 18585.943} C_VEL
LIN {X 0,Y 504.682,Z 249.854,A -85,B 0,C 180,E1 18582.499,E2 18582.499} C_VEL
LIN {X 0,Y 504.707,Z 249.866,A -85,B 0,C 180,E1 18579.049,E2 18579.049} C_VEL
LIN {X 0,Y 504.702,Z 249.869,A -85,B 0,C 180,E1 18575.483,E2 18575.483} C_VEL
LIN {X 0,Y 504.707,Z 249.865,A -85,B 0,C 180,E1 18571.935,E2 18571.935} C_VEL
LIN {X 0,Y 504.696,Z 249.864,A -85,B 0,C 180,E1 18568.39,E2 18568.39} C_VEL
LIN {X 0,Y 504.706,Z 249.865,A -85,B 0,C 180,E1 18564.834,E2 18564.834} C_VEL
LIN {X 0,Y 504.692,Z 249.864,A -85,B 0,C 180,E1 18561.379,E2 18561.379} C_VEL
LIN {X 0,Y 504.703,Z 249.864,A -85,B 0,C 180,E1 18557.883,E2 18557.883} C_VEL
LIN {X 0,Y 504.704,Z 249.863,A -85,B 0,C 180,E1 18554.338,E2 18554.338} C_VEL
LIN {X 0,Y 504.697,Z 249.858,A -85,B 0,C 180,E1 18550.849,E2 18550.849} C_VEL
LIN {X 0,Y 504.68,Z 249.867,A -85,B 0,C 180,E1 18547.4,E2 18547.4} C_VEL
LIN {X 0,Y 504.704,Z 249.864,A -85,B 0,C 180,E1 18543.977,E2 18543.977} C_VEL
LIN {X 0,Y 504.71,Z 249.863,A -85,B 0,C 180,E1 18540.455,E2 18540.455} C_VEL
LIN {X 0,Y 504.67,Z 249.869,A -85,B 0,C 180,E1 18537.048,E2 18537.048} C_VEL
LIN {X 0,Y 504.671,Z 249.867,A -85,B 0,C 180,E1 18533.517,E2 18533.517} C_VEL
LIN {X 0,Y 504.71,Z 249.864,A -85,B 0,C 180,E1 18530.077,E2 18530.077} C_VEL
LIN {X 0,Y 504.676,Z 249.87,A -85,B 0,C 180,E1 18526.598,E2 18526.598} C_VEL
LIN {X 0,Y 504.653,Z 249.873,A -85,B 0,C 180,E1 18523.13,E2 18523.13} C_VEL
LIN {X 0,Y 504.684,Z 249.869,A -85,B 0,C 180,E1 18519.716,E2 18519.716} C_VEL
LIN {X 0,Y 504.671,Z 249.86,A -85,B 0,C 180,E1 18516.41,E2 18516.41} C_VEL
LIN {X 0,Y 504.685,Z 250.165,A -85,B 0,C 180,E1 18515.073,E2 18515.073} C_VEL
LIN {X 0,Y 512.247,Z 268.222,A -85,B 0,C 180,E1 18512.572,E2 18512.572} C_VEL
LIN {X 0,Y 516.442,Z 279.239,A -85,B 0,C 180,E1 18511.18,E2 18511.18} C_VEL
LIN {X 0,Y 515.325,Z 299.978,A -85,B 0,C 180,E1 18509.448,E2 18509.448} C_VEL
LIN {X 0,Y 518.6,Z 318.295,A -85,B 0,C 180,E1 18508.863,E2 18508.863} C_VEL
LIN {X 0,Y 516.875,Z 432.639,A -85,B 0,C 180,E1 18507.081,E2 18507.081} C_VEL
LIN {X 0,Y 515.971,Z 440.329,A -85,B 0,C 180,E1 18507.022,E2 18507.022} C_VEL
LIN {X 0,Y 510.476,Z 460.847,A -85,B 0,C 180,E1 18507.095,E2 18507.095} C_VEL
LIN {X 0,Y 509.717,Z 467.45,A -85,B 0,C 180,E1 18507.041,E2 18507.041} C_VEL
LIN {X 0,Y 508.169,Z 563.242,A -85,B 0,C 180,E1 18505.51,E2 18505.51} C_VEL
LIN {X 0,Y 507.416,Z 584.029,A -85,B 0,C 180,E1 18504.966,E2 18504.966} C_VEL
LIN {X 0,Y 506.484,Z 603.482,A -85,B 0,C 180,E1 18504.246,E2 18504.246} C_VEL
LIN {X 0,Y 505.312,Z 623.03,A -85,B 0,C 180,E1 18503.306,E2 18503.306} C_VEL
LIN {X 0,Y 503.99,Z 642.182,A -85,B 0,C 180,E1 18502.148,E2 18502.148} C_VEL
LIN {X 0,Y 502.696,Z 659.497,A -85,B 0,C 180,E1 18500.87,E2 18500.87} C_VEL
LIN {X 0,Y 501.33,Z 676.512,A -85,B 0,C 180,E1 18499.366,E2 18499.366} C_VEL
LIN {X 0,Y 499.987,Z 692.885,A -85,B 0,C 180,E1 18497.632,E2 18497.632} C_VEL
LIN {X 0,Y 498.66,Z 710.312,A -85,B 0,C 180,E1 18495.432,E2 18495.432} C_VEL
LIN {X 0,Y 497.805,Z 723.146,A -85,B 0,C 180,E1 18493.527,E2 18493.527} C_VEL
LIN {X 0,Y 497.062,Z 735.78,A -85,B 0,C 180,E1 18491.284,E2 18491.284} C_VEL
LIN {X 0,Y 496.552,Z 746.05,A -85,B 0,C 180,E1 18489.07,E2 18489.07} C_VEL
LIN {X 0,Y 496.233,Z 754.346,A -85,B 0,C 180,E1 18486.881,E2 18486.881} C_VEL
LIN {X 0,Y 496.029,Z 761.484,A -85,B 0,C 180,E1 18484.502,E2 18484.502} C_VEL
LIN {X 0,Y 495.943,Z 766.75,A -85,B 0,C 180,E1 18482.143,E2 18482.143} C_VEL
LIN {X 0,Y 495.92,Z 770.226,A -85,B 0,C 180,E1 18479.868,E2 18479.868} C_VEL
LIN {X 0,Y 495.912,Z 772.124,A -85,B 0,C 180,E1 18477.489,E2 18477.489} C_VEL
LIN {X 0,Y 495.912,Z 772.348,A -85,B 0,C 180,E1 18475.144,E2 18475.144} C_VEL
LIN {X 0,Y 495.912,Z 770.949,A -85,B 0,C 180,E1 18472.776,E2 18472.776} C_VEL
LIN {X 0,Y 495.929,Z 768.119,A -85,B 0,C 180,E1 18470.538,E2 18470.538} C_VEL
LIN {X 0,Y 495.993,Z 763.507,A -85,B 0,C 180,E1 18468.209,E2 18468.209} C_VEL
LIN {X 0,Y 496.145,Z 757.212,A -85,B 0,C 180,E1 18465.908,E2 18465.908} C_VEL
LIN {X 0,Y 496.421,Z 749.232,A -85,B 0,C 180,E1 18463.631,E2 18463.631} C_VEL
LIN {X 0,Y 496.865,Z 739.432,A -85,B 0,C 180,E1 18461.375,E2 18461.375} C_VEL
LIN {X 0,Y 497.484,Z 728.292,A -85,B 0,C 180,E1 18459.254,E2 18459.254} C_VEL
LIN {X 0,Y 498.286,Z 715.879,A -85,B 0,C 180,E1 18457.264,E2 18457.264} C_VEL
LIN {X 0,Y 499.318,Z 701.204,A -85,B 0,C 180,E1 18455.286,E2 18455.286} C_VEL
LIN {X 0,Y 500.584,Z 685.215,A -85,B 0,C 180,E1 18453.436,E2 18453.436} C_VEL
LIN {X 0,Y 501.874,Z 669.243,A -85,B 0,C 180,E1 18451.885,E2 18451.885} C_VEL
LIN {X 0,Y 503.171,Z 652.492,A -85,B 0,C 180,E1 18450.514,E2 18450.514} C_VEL
LIN {X 0,Y 504.49,Z 634.119,A -85,B 0,C 180,E1 18449.263,E2 18449.263} C_VEL
LIN {X 0,Y 505.699,Z 615.744,A -85,B 0,C 180,E1 18448.245,E2 18448.245} C_VEL
LIN {X 0,Y 506.774,Z 595.614,A -85,B 0,C 180,E1 18447.365,E2 18447.365} C_VEL
LIN {X 0,Y 507.657,Z 575.279,A -85,B 0,C 180,E1 18446.713,E2 18446.713} C_VEL
LIN {X 0,Y 508.22,Z 554.719,A -85,B 0,C 180,E1 18446.265,E2 18446.265} C_VEL
LIN {X 0,Y 511.769,Z 318.822,A -85,B 0,C 180,E1 18442.582,E2 18442.582} C_VEL
LIN {X 0,Y 508.175,Z 298.992,A -85,B 0,C 180,E1 18441.914,E2 18441.914} C_VEL
LIN {X 0,Y 509.021,Z 281.613,A -85,B 0,C 180,E1 18440.413,E2 18440.413} C_VEL
LIN {X 0,Y 502.184,Z 264.207,A -85,B 0,C 180,E1 18438.167,E2 18438.167} C_VEL
LIN {X 0,Y 496.812,Z 251.185,A -85,B 0,C 180,E1 18436.353,E2 18436.353} C_VEL
LIN {X 0,Y 496.754,Z 250.826,A -85,B 0,C 180,E1 18435.668,E2 18435.668} C_VEL
LIN {X 0,Y 496.762,Z 250.825,A -85,B 0,C 180,E1 18432.176,E2 18432.176} C_VEL
LIN {X 0,Y 496.772,Z 250.855,A -85,B 0,C 180,E1 18428.637,E2 18428.637} C_VEL
LIN {X 0,Y 496.747,Z 250.837,A -85,B 0,C 180,E1 18425.124,E2 18425.124} C_VEL
LIN {X 0,Y 496.765,Z 250.85,A -85,B 0,C 180,E1 18421.586,E2 18421.586} C_VEL
LIN {X 0,Y 496.765,Z 250.848,A -85,B 0,C 180,E1 18418.04,E2 18418.04} C_VEL
LIN {X 0,Y 496.766,Z 250.845,A -85,B 0,C 180,E1 18414.433,E2 18414.433} C_VEL
LIN {X 0,Y 496.744,Z 250.849,A -85,B 0,C 180,E1 18410.951,E2 18410.951} C_VEL
LIN {X 0,Y 496.765,Z 250.856,A -85,B 0,C 180,E1 18407.445,E2 18407.445} C_VEL
LIN {X 0,Y 496.766,Z 250.852,A -85,B 0,C 180,E1 18403.902,E2 18403.902} C_VEL
LIN {X 0,Y 496.763,Z 250.844,A -85,B 0,C 180,E1 18400.288,E2 18400.288} C_VEL
LIN {X 0,Y 496.744,Z 250.845,A -85,B 0,C 180,E1 18396.711,E2 18396.711} C_VEL
LIN {X 0,Y 496.761,Z 250.857,A -85,B 0,C 180,E1 18393.147,E2 18393.147} C_VEL
LIN {X 0,Y 496.764,Z 250.845,A -85,B 0,C 180,E1 18389.603,E2 18389.603} C_VEL
LIN {X 0,Y 496.756,Z 250.847,A -85,B 0,C 180,E1 18386.147,E2 18386.147} C_VEL
LIN {X 0,Y 496.745,Z 250.857,A -85,B 0,C 180,E1 18382.608,E2 18382.608} C_VEL
LIN {X 0,Y 496.766,Z 250.843,A -85,B 0,C 180,E1 18379.151,E2 18379.151} C_VEL
LIN {X 0,Y 496.769,Z 250.852,A -85,B 0,C 180,E1 18375.526,E2 18375.526} C_VEL
LIN {X 0,Y 496.751,Z 250.852,A -85,B 0,C 180,E1 18371.964,E2 18371.964} C_VEL
LIN {X 0,Y 496.742,Z 250.845,A -85,B 0,C 180,E1 18368.448,E2 18368.448} C_VEL
LIN {X 0,Y 496.767,Z 250.857,A -85,B 0,C 180,E1 18364.951,E2 18364.951} C_VEL
LIN {X 0,Y 496.768,Z 250.847,A -85,B 0,C 180,E1 18361.383,E2 18361.383} C_VEL
LIN {X 0,Y 496.743,Z 250.843,A -85,B 0,C 180,E1 18357.923,E2 18357.923} C_VEL
LIN {X 0,Y 496.745,Z 250.854,A -85,B 0,C 180,E1 18354.339,E2 18354.339} C_VEL
LIN {X 0,Y 496.768,Z 250.851,A -85,B 0,C 180,E1 18350.85,E2 18350.85} C_VEL
LIN {X 0,Y 496.763,Z 250.84,A -85,B 0,C 180,E1 18347.326,E2 18347.326} C_VEL
LIN {X 0,Y 496.738,Z 250.849,A -85,B 0,C 180,E1 18343.872,E2 18343.872} C_VEL
LIN {X 0,Y 496.757,Z 250.856,A -85,B 0,C 180,E1 18340.358,E2 18340.358} C_VEL
LIN {X 0,Y 496.771,Z 250.854,A -85,B 0,C 180,E1 18336.891,E2 18336.891} C_VEL
LIN {X 0,Y 496.75,Z 250.855,A -85,B 0,C 180,E1 18333.329,E2 18333.329} C_VEL
LIN {X 0,Y 496.738,Z 250.859,A -85,B 0,C 180,E1 18329.787,E2 18329.787} C_VEL
LIN {X 0,Y 496.761,Z 250.859,A -85,B 0,C 180,E1 18326.253,E2 18326.253} C_VEL
LIN {X 0,Y 496.772,Z 250.853,A -85,B 0,C 180,E1 18322.654,E2 18322.654} C_VEL
LIN {X 0,Y 496.746,Z 250.852,A -85,B 0,C 180,E1 18319.143,E2 18319.143} C_VEL
LIN {X 0,Y 496.733,Z 250.824,A -85,B 0,C 180,E1 18315.534,E2 18315.534} C_VEL
LIN {X 0,Y 496.815,Z 251.166,A -85,B 0,C 180,E1 18314.689,E2 18314.689} C_VEL
LIN {X 0,Y 498.167,Z 254.464,A -85,B 0,C 180,E1 18314.231,E2 18314.231} C_VEL
LIN {X 0,Y 506.053,Z 271.438,A -85,B 0,C 180,E1 18312.105,E2 18312.105} C_VEL
LIN {X 0,Y 513.146,Z 287.172,A -85,B 0,C 180,E1 18310.285,E2 18310.285} C_VEL
LIN {X 0,Y 512.489,Z 302.7,A -85,B 0,C 180,E1 18309.247,E2 18309.247} C_VEL
LIN {X 0,Y 515.633,Z 323.256,A -85,B 0,C 180,E1 18308.637,E2 18308.637} C_VEL
LIN {X 0,Y 512.653,Z 540.524,A -85,B 0,C 180,E1 18305.259,E2 18305.259} C_VEL
LIN {X 0,Y 511.652,Z 609.697,A -85,B 0,C 180,E1 18304.168,E2 18304.168} C_VEL
LIN {X 0,Y 510.831,Z 630.246,A -85,B 0,C 180,E1 18303.653,E2 18303.653} C_VEL
LIN {X 0,Y 509.697,Z 652.426,A -85,B 0,C 180,E1 18302.882,E2 18302.882} C_VEL
LIN {X 0,Y 508.489,Z 672.195,A -85,B 0,C 180,E1 18301.999,E2 18301.999} C_VEL
LIN {X 0,Y 507.033,Z 691.765,A -85,B 0,C 180,E1 18300.909,E2 18300.909} C_VEL
LIN {X 0,Y 505.463,Z 711.921,A -85,B 0,C 180,E1 18299.554,E2 18299.554} C_VEL
LIN {X 0,Y 503.93,Z 730.062,A -85,B 0,C 180,E1 18298.112,E2 18298.112} C_VEL
LIN {X 0,Y 502.36,Z 748.135,A -85,B 0,C 180,E1 18296.408,E2 18296.408} C_VEL
LIN {X 0,Y 500.87,Z 765.175,A -85,B 0,C 180,E1 18294.531,E2 18294.531} C_VEL
LIN {X 0,Y 499.611,Z 780.337,A -85,B 0,C 180,E1 18292.595,E2 18292.595} C_VEL
LIN {X 0,Y 498.484,Z 794.874,A -85,B 0,C 180,E1 18290.425,E2 18290.425} C_VEL
LIN {X 0,Y 497.624,Z 807.192,A -85,B 0,C 180,E1 18288.265,E2 18288.265} C_VEL
LIN {X 0,Y 496.93,Z 818.788,A -85,B 0,C 180,E1 18285.88,E2 18285.88} C_VEL
LIN {X 0,Y 496.464,Z 828.435,A -85,B 0,C 180,E1 18283.509,E2 18283.509} C_VEL
LIN {X 0,Y 496.159,Z 836.438,A -85,B 0,C 180,E1 18281.067,E2 18281.067} C_VEL
LIN {X 0,Y 495.997,Z 842.894,A -85,B 0,C 180,E1 18278.578,E2 18278.578} C_VEL
LIN {X 0,Y 495.935,Z 847.638,A -85,B 0,C 180,E1 18276.133,E2 18276.133} C_VEL
LIN {X 0,Y 495.906,Z 850.675,A -85,B 0,C 180,E1 18273.698,E2 18273.698} C_VEL
LIN {X 0,Y 495.91,Z 852.282,A -85,B 0,C 180,E1 18271.154,E2 18271.154} C_VEL
LIN {X 0,Y 495.91,Z 852.281,A -85,B 0,C 180,E1 18268.844,E2 18268.844} C_VEL
LIN {X 0,Y 495.907,Z 850.671,A -85,B 0,C 180,E1 18266.3,E2 18266.3} C_VEL
LIN {X 0,Y 495.936,Z 847.63,A -85,B 0,C 180,E1 18263.865,E2 18263.865} C_VEL
LIN {X 0,Y 495.997,Z 843.142,A -85,B 0,C 180,E1 18261.537,E2 18261.537} C_VEL
LIN {X 0,Y 496.147,Z 836.878,A -85,B 0,C 180,E1 18259.079,E2 18259.079} C_VEL
LIN {X 0,Y 496.422,Z 829.252,A -85,B 0,C 180,E1 18256.725,E2 18256.725} C_VEL
LIN {X 0,Y 496.867,Z 819.807,A -85,B 0,C 180,E1 18254.355,E2 18254.355} C_VEL
LIN {X 0,Y 497.539,Z 808.449,A -85,B 0,C 180,E1 18251.971,E2 18251.971} C_VEL
LIN {X 0,Y 498.435,Z 795.624,A -85,B 0,C 180,E1 18249.693,E2 18249.693} C_VEL
LIN {X 0,Y 499.541,Z 781.169,A -85,B 0,C 180,E1 18247.523,E2 18247.523} C_VEL
LIN {X 0,Y 500.806,Z 765.951,A -85,B 0,C 180,E1 18245.561,E2 18245.561} C_VEL
LIN {X 0,Y 502.26,Z 749.297,A -85,B 0,C 180,E1 18243.708,E2 18243.708} C_VEL
LIN {X 0,Y 503.789,Z 731.657,A -85,B 0,C 180,E1 18242.029,E2 18242.029} C_VEL
LIN {X 0,Y 505.352,Z 713.217,A -85,B 0,C 180,E1 18240.542,E2 18240.542} C_VEL
LIN {X 0,Y 506.891,Z 693.736,A -85,B 0,C 180,E1 18239.21,E2 18239.21} C_VEL
LIN {X 0,Y 508.412,Z 673.36,A -85,B 0,C 180,E1 18238.06,E2 18238.06} C_VEL
LIN {X 0,Y 509.657,Z 653.19,A -85,B 0,C 180,E1 18237.149,E2 18237.149} C_VEL
LIN {X 0,Y 510.813,Z 630.75,A -85,B 0,C 180,E1 18236.361,E2 18236.361} C_VEL
LIN {X 0,Y 511.619,Z 610.587,A -85,B 0,C 180,E1 18235.852,E2 18235.852} C_VEL
LIN {X 0,Y 512.294,Z 566.534,A -85,B 0,C 180,E1 18235.143,E2 18235.143} C_VEL
LIN {X 0,Y 515.16,Z 347.308,A -85,B 0,C 180,E1 18231.762,E2 18231.762} C_VEL
LIN {X 0,Y 515.311,Z 320.92,A -85,B 0,C 180,E1 18231.332,E2 18231.332} C_VEL
LIN {X 0,Y 512.235,Z 301.506,A -85,B 0,C 180,E1 18230.733,E2 18230.733} C_VEL
LIN {X 0,Y 512.851,Z 286.734,A -85,B 0,C 180,E1 18229.715,E2 18229.715} C_VEL
LIN {X 0,Y 501.735,Z 262.079,A -85,B 0,C 180,E1 18226.834,E2 18226.834} C_VEL
LIN {X 0,Y 497.899,Z 254.055,A -85,B 0,C 180,E1 18225.8,E2 18225.8} C_VEL
LIN {X 0,Y 496.812,Z 251.152,A -85,B 0,C 180,E1 18225.404,E2 18225.404} C_VEL
LIN {X 0,Y 496.758,Z 250.855,A -85,B 0,C 180,E1 18224.141,E2 18224.141} C_VEL
LIN {X 0,Y 496.748,Z 250.858,A -85,B 0,C 180,E1 18220.552,E2 18220.552} C_VEL
LIN {X 0,Y 496.765,Z 250.856,A -85,B 0,C 180,E1 18217,E2 18217} C_VEL
LIN {X 0,Y 496.763,Z 250.857,A -85,B 0,C 180,E1 18213.47,E2 18213.47} C_VEL
